# B&R Automation Studio project Embraco_PracoviskoPopisovaniaLaserom
Automation Studio 4.7.6.114 SP; technology packages: mapp 5.13.1

## Configuration Config1

CPU X20CP0484, AutomationRuntime D4.73, Build 6.3.0, Safety 1.10, Vc V4.72.4

### Task classes (Cpu.sw)
```
Cyclic#1 (cycle 2000 us, tolerance 0 us):
  CheckerKom <- Komunikacia_Checker.CheckerKomunikacia.prg
  MeranieTak <- Program.MeranieTaktime.prg
Cyclic#3 (cycle 50000 us, tolerance 50000 us):
  VstupnyOdd <- Program.VstupnyOddelovac.prg
  Popisovani <- Program.Popisovanie.prg
  Checker <- Program.Checker.prg
Cyclic#4 (cycle 100000 us, tolerance 100000 us):
  Main <- Program.Main.prg
  Poruchy_Si <- Program.Poruchy_Signalizacie.prg
  OvladanieG <- HMI.OvladanieGrafiky.prg
  Vycitanie_ <- Komunikacia_Laser.Vycitanie_casu.prg
  Ethernetov <- Komunikacia_Laser.EthernetovaKomunikacia.prg
Cyclic#5 (cycle 200000 us, tolerance 200000 us):
  Receptury <- Receptury.Receptury.prg
  Prihlasova <- PrihlasovaciSystem.PrihlasovaciSystem.prg
  Blikanie20 <- Blikace.Blikanie200ms.prg
Cyclic#6 (cycle 500000 us, tolerance 500000 us):
  Blikanie50 <- Blikace.Blikanie500ms.prg
Cyclic#7 (cycle 1000000 us, tolerance 1000000 us):
  Blikanie1s <- Blikace.Blikanie1s.prg
DataObjects: assl1
VcDataObjects: Visu <- HMI.Visu.dob
Binaries: vcfile, vcnet, vcbclass, vcfntttf, Visu01, arsvcreg, vcshared, vcpkat, vcpfgen, TCData, vcmgr, vctcal, vcalarm, vcdsloc, vcpdsw, vcdsint, vcrt, arial, udbdef, vcgclass, vcpdvnc, Visu02, vccdt, vccbmp, vccstr, vccbtn, vccline, vcclbox, arialbd, vccnum, vccalarm, vccbar, vcctext, Visu03, vccovl, vccshape, vcchspot, asnxdb1, iomap, Config_2, sysconf, Config, ashwac, Config_1, ashwd, asfw, User, arconfig, Role
Libraries: AsSafety, FileIO, DataObj, AsXml, standard, runtime, astime, AsBrStr, IecCheck, sys_lib, SC, MpRecipe, MpBase, AsTCP, AsMath, asieccon, vcresman
```

### Hardware
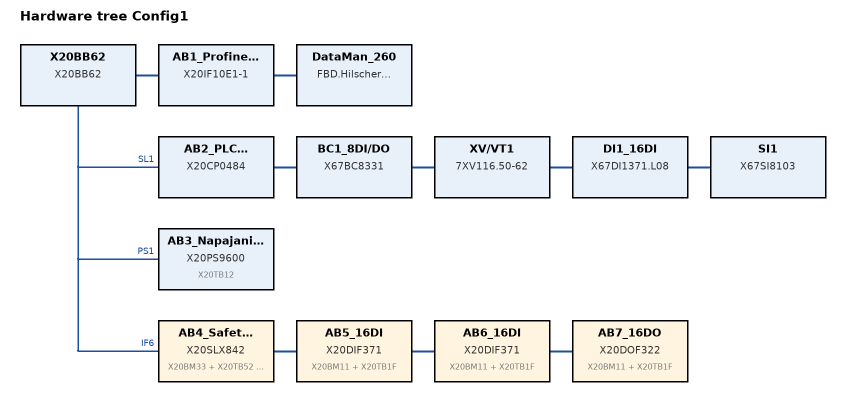
```
AB1_ProfinetMaster : X20IF10E1-1 v1.3.0.0  [SS -> X20BB62.SS1]
  Connector IF1:
    DtmRef = FBDIF.Hilscher.PNIOControllerDTM2.NETX 100 RE/PNM
    DtmId = eaec8113-ff32-47e2-8a6f-5691c0f842d4
  ConfigFile = AB1_ProfinetMaster.dtm
  ConfigModule = asnxdb1
AB2_PLC_X20CP0484 : X20CP0484 v1.4.2.0  [SL -> X20BB62.SL1]
  Connector IF2:
    ActivateDevice = 1
    Mode = Manual
    InternetAddress = 192.168.1.2
    SubnetMask = 255.255.255.0
    InaNodeNumber = 0
    Vnc1
    VncVcObjectName1 = Visu
    VncKeyMappingFile1 = VC\PS2-Keyboard.dis
    VncMaxConnections1 = 2
    VncRefreshRate1 = 100
  ConfigurationID = Embraco_PracoviskoPopisovaniaLaserom_Config1
  UserPartitionSize = 500
  UserRamSize = 10000
  RemMemSize = 20000
  PermanentPvSize = 8000
  TimerDeviceType = EPLX2X
  TimerDevice = AB2_PLC_X20CP0484.IF3
  TaskClassIdleTime = 2000
  Cyclic1Duration = 2000
  Cyclic1Tolerance = 0
  Cyclic2Duration = 10000
  Cyclic2Tolerance = 0
  Cyclic3Duration = 50000
  Cyclic3Tolerance = 50000
  Cyclic4Duration = 100000
  Cyclic4Tolerance = 100000
  Cyclic5Duration = 200000
  Cyclic5Tolerance = 200000
  Cyclic6Duration = 500000
  Cyclic6Tolerance = 500000
  Cyclic7Duration = 1000000
  Cyclic7Tolerance = 1000000
  Cyclic8Duration = 10000
  Cyclic8Tolerance = 30000000
  FileDevice1
  FileDeviceName1 = HDD
  FileDevicePath1 = F:\
  TimeZone = 145
  ActivateSntpServer = 1
  FtpUser1
  FtpUsername1 = admin
  FtpUserPassword1 = ZFxZtXmikHeuYrBmUWmLP4sX8b0VA9Bjt2tGuquGkoo=
  FtpUserSalt1 = qbFABSSZ
  FTPAccessRight1 = 0
AB3_NapajaniePLC : X20PS9600 v1.5.0.0  [PS -> X20BB62.PS1; SS1 -> X20TB12.SS]
AB4_SafetyMaster : X20SLX842 v1.10.12.1  [SS1 -> X20TB52.SS; SS2 -> X20TB52a.SS; SL -> X20BM33.SL1]
  Supervision = off
  SafeProject = SafeLOGIC-1
  SafeDesigner = 4.4.0.0
  DigitalOutput01 = viaSafeLOGIC
  DigitalOutput02 = viaSafeLOGIC
  DigitalOutput03 = viaSafeLOGIC
  DigitalOutput04 = viaSafeLOGIC
  DigitalOutput05 = viaSafeLOGIC
  DigitalOutput06 = viaSafeLOGIC
  UnsafeOutputBOOLs = 32
  UnsafeInputBOOLs = 32
AB5_16DI : X20DIF371 v1.1.0.0  [SS1 -> X20TB1F.SS; SL -> X20BM11.SL1]
  Supervision = off
AB6_16DI : X20DIF371 v1.1.0.0  [SS1 -> X20TB1F1.SS; SL -> X20BM11a.SL1]
  Supervision = off
AB7_16DO : X20DOF322 v1.4.0.0  [SS1 -> X20TB1F2.SS; SL -> X20BM11b.SL1]
  Supervision = off
BC1_8DI/DO : X67BC8331 v2.11.1.0  [PLK1 -> AB2_PLC_X20CP0484.IF3 [Cable Type=PowerlinkCable, Length=10, Version=1.0.0.2]]
DI1_16DI : X67DI1371.L08 v1.1.0.0  [X2X1 -> XV/VT1.X2X2 [Cable Type=X2XCable, Length=10, Version=1.0.0.2]]
  Supervision = off
DataMan_260 : FBD.Hilscher.PNIOGenDevDTM2.DataMan 260 v5.5.0 (OrderNumber=DataMan 260, VendorAddress=dataman)  [PN1 -> AB1_ProfinetMaster.IF1]
  DtmId = 4941676e-6e57-439f-abc9-d0f1f6497b10
  ChannelBlocks_47615121-fe6e-4591-b3b6-8465b3212ca9  // Acquisition Control <Slot 1>
  IO_OutputImage_47615121-fe6e-4591-b3b6-8465b3212ca9  // 1 Byte(s)
  ChannelBlocks_d194d4db-42e7-41e5-a767-b87b0401a075  // Acquisition Status <Slot 2>
  IO_InputImage_d194d4db-42e7-41e5-a767-b87b0401a075  // 3 Byte(s)
  ChannelBlocks_1f3ce926-3699-4ff7-ae20-f41f99e8e1a7  // Results Control <Slot 3>
  IO_OutputImage_1f3ce926-3699-4ff7-ae20-f41f99e8e1a7  // 1 Byte(s)
  ChannelBlocks_275960ff-423a-4b85-9ae8-7b4c1d1c8472  // Results Status <Slot 4>
  IO_InputImage_275960ff-423a-4b85-9ae8-7b4c1d1c8472  // 1 Byte(s)
  ChannelBlocks_ec76be99-af22-40a4-a52c-c51730de08a4  // Soft Event Control <Slot 5>
  IO_InputImage_ec76be99-af22-40a4-a52c-c51730de08a4  // 1 Byte(s)
  IO_OutputImage_ec76be99-af22-40a4-a52c-c51730de08a4  // 1 Byte(s)
  ChannelBlocks_de08c721-900e-43fb-8e68-4cff8c152ca9  // User Data - 64 bytes <Slot 6>
  IO_OutputImage_de08c721-900e-43fb-8e68-4cff8c152ca9  // 68 Byte(s)
  ChannelBlocks_b5868303-eee8-413e-96c2-c1ebf3a28649  // Result Data - 64 bytes <Slot 7>
  IO_InputImage_b5868303-eee8-413e-96c2-c1ebf3a28649  // 72 Byte(s)
SI1 : X67SI8103 v1.10.12.0  [X2X1 -> DI1_16DI.X2X2 [Cable Type=X2XCable, Length=10, Version=1.0.0.2]]
  Supervision = off
X20BB62 : X20BB62 v1.1.1.0
X20BM11 : X20BM11 v1.0.0.1  [X2X1 -> X20BM33.X2X2]
X20BM11a : X20BM11 v1.0.0.1  [X2X1 -> X20BM11.X2X2]
X20BM11b : X20BM11 v1.0.0.1  [X2X1 -> X20BM11a.X2X2]
X20BM33 : X20BM33 v1.0.0.6  [X2X1 -> X20BB62.IF6]
X20TB12 : X20TB12 v1.0.0.0
X20TB1F : X20TB1F v1.0.0.0
X20TB1F1 : X20TB1F v1.0.0.0
X20TB1F2 : X20TB1F v1.0.0.0
X20TB52 : X20TB52 v1.0.0.2
X20TB52a : X20TB52 v1.0.0.2
XV/VT1 : 7XV116.50-62 v1.2.0.0  [X2X1 -> BC1_8DI/DO.IF1 [Cable Type=X2XCable, Length=10, Version=1.0.0.2]]
  Supervision = off
```

### Cpu.per - AB2_PLC_X20CP0484/Cpu.per
```iecst
VAR_CONFIG
	Stav_StatorPopisany AT %MX0; (* *)
END_VAR
```

### IoMap.iom - AB2_PLC_X20CP0484/IoMap.iom
```iecst
VAR_CONFIG
	Cyclic#1.Safety.IN.CS_Panel_KanalA AT %IX."AB4_SafetyMaster".SafeDigitalInput01;
	Cyclic#1.Safety.IN.CS_Panel_KanalB AT %IX."AB4_SafetyMaster".SafeDigitalInput02;
	Cyclic#1.Safety.IN.CS_Checker_KanalA AT %IX."AB4_SafetyMaster".SafeDigitalInput03;
	Cyclic#1.Safety.IN.CS_Checker_KanalB AT %IX."AB4_SafetyMaster".SafeDigitalInput04;
	Cyclic#1.Safety.IN.VyblokovanieZamkov_KanalA AT %IX."AB4_SafetyMaster".SafeDigitalInput05;
	Cyclic#1.Safety.IN.VyblokovanieZamkov_KanalB AT %IX."AB4_SafetyMaster".SafeDigitalInput06;
	Cyclic#1.Safety.OUT.Zona_CS AT %IX."AB4_SafetyMaster".PhysicalStateChannel01;
	Cyclic#1.Safety.OUT.Zona_VnutroBunky AT %IX."AB4_SafetyMaster".PhysicalStateChannel02;
	Cyclic#1.Safety.OUT.Zona_Laser AT %IX."AB4_SafetyMaster".PhysicalStateChannel03;
	Cyclic#1.Safety.OUT.Zona_ExternyCS_KanalA AT %IX."AB4_SafetyMaster".PhysicalStateChannel05;
	Cyclic#1.Safety.OUT.Zona_ExternyCS_KanalB AT %IX."AB4_SafetyMaster".PhysicalStateChannel06;
	Cyclic#1.Safety.RESET_ZonyCS AT %QX."AB4_SafetyMaster".BOOL101;
	Cyclic#1.Safety.RESET_ZonyLaser AT %QX."AB4_SafetyMaster".BOOL102;
	Cyclic#1.Safety.RESET_ZonyVnutroBunky AT %QX."AB4_SafetyMaster".BOOL103;
	Cyclic#1.Safety.IN.ZonaCS_SpatnaVezba AT %QX."AB4_SafetyMaster".BOOL104;
	Cyclic#1.Safety.IN.ZonaLaser_SpatnaVezba AT %QX."AB4_SafetyMaster".BOOL105;
	Cyclic#1.Safety.IN.ZonaVnutroBunky_SpatnaVezba AT %QX."AB4_SafetyMaster".BOOL106;
	Cyclic#1.Zariadenie.IN.TlakVzduchu_OK AT %QX."AB4_SafetyMaster".BOOL107;
	Cyclic#1.Safety.STAV.SafetyPLC_Nabehlo AT %IX."AB4_SafetyMaster".BOOL001;
	Cyclic#1.Safety.STAV.CS_Panel_Odblokov AT %IX."AB4_SafetyMaster".BOOL002;
	Cyclic#1.Safety.STAV.CS_Checker_Odblokov AT %IX."AB4_SafetyMaster".BOOL003;
	Cyclic#1.Safety.STAV.DvereBunky_Zamknute AT %IX."AB4_SafetyMaster".BOOL004;
	Cyclic#1.Safety.STAV.SnimacKrytuLasera_Aktivny AT %IX."AB4_SafetyMaster".BOOL005;
	Cyclic#1.Safety.STAV.SnimacStatorPodLaserom_Aktivny AT %IX."AB4_SafetyMaster".BOOL006;
	Cyclic#1.Safety.STAV.VyblokovanieZamkov_Aktivne AT %IX."AB4_SafetyMaster".BOOL007;
	Cyclic#1.Safety.STAV.ZonaCS_Aktivna AT %IX."AB4_SafetyMaster".BOOL008;
	Cyclic#1.Safety.STAV.ZonaLaser_Aktivna AT %IX."AB4_SafetyMaster".BOOL009;
	Cyclic#1.Safety.STAV.ZonaVnutroBunky_Aktivna AT %IX."AB4_SafetyMaster".BOOL010;
	Cyclic#1.Safety.IN.DvereBunky_KanalA AT %IX."SI1".SafeDigitalInput01;
	Cyclic#1.Safety.IN.DvereBunky_KanalB AT %IX."SI1".SafeDigitalInput02;
	Cyclic#1.Safety.IN.StatorPodLaserom_KanalA AT %IX."SI1".SafeDigitalInput03;
	Cyclic#1.Safety.IN.StatorPodLaserom_KanalB AT %IX."SI1".SafeDigitalInput04;
	Cyclic#1.Safety.IN.KrytLasera_KanalA AT %IX."SI1".SafeDigitalInput05;
	Cyclic#1.Safety.IN.KrytLasera_KanalB AT %IX."SI1".SafeDigitalInput06;
	Cyclic#1.Safety.OUT.DvereBunky_Zamkni AT %QX."SI1".DigitalOutput01;
	Cyclic#1.Zariadenie.IN.PrepatovaOchrana_OK AT %IX."AB5_16DI".DigitalInput01;
	Cyclic#1.Safety.IN.ZdvihZdvizky_SpatnaVezba AT %QX."AB4_SafetyMaster".BOOL108;
	Cyclic#1.Zariadenie.IN.NapajanieOdsavania_OK AT %IX."AB5_16DI".DigitalInput02;
	Cyclic#1.Zariadenie.IN.NapajanieLasera_OK AT %IX."AB5_16DI".DigitalInput03;
	Cyclic#1.Zariadenie.IN.TlacitkoSTART AT %IX."AB5_16DI".DigitalInput04;
	Cyclic#1.Zariadenie.IN.TlacitkoSTOP AT %IX."AB5_16DI".DigitalInput05;
	Cyclic#1.Zariadenie.IN.TlacitkoRESET_CS AT %IX."AB5_16DI".DigitalInput06;
	Cyclic#1.Zariadenie.IN.TlakVzduchu_OK AT %IX."AB5_16DI".DigitalInput07;
	Cyclic#1.Checker.IN.TlacitkoBANNER AT %IX."AB5_16DI".DigitalInput08;
	Cyclic#1.Safety.IN.ZdvihZdvizky_SpatnaVezba AT %IX."AB5_16DI".DigitalInput09;
	Cyclic#1.Safety.IN.ZonaCS_SpatnaVezba AT %IX."AB5_16DI".DigitalInput10;
	Cyclic#1.Safety.IN.ZonaVnutroBunky_SpatnaVezba AT %IX."AB5_16DI".DigitalInput11;
	Cyclic#1.Safety.IN.ZonaLaser_SpatnaVezba AT %IX."AB5_16DI".DigitalInput12;
	Cyclic#1.Popisovanie.IN.Laser_StavREADY AT %IX."AB5_16DI".DigitalInput13;
	Cyclic#1.Popisovanie.IN.Laser_StavEND AT %IX."AB5_16DI".DigitalInput14;
	Cyclic#1.Popisovanie.IN.Laser_StavBUSY AT %IX."AB5_16DI".DigitalInput15;
	Cyclic#1.Popisovanie.IN.Laser_STARTUP AT %IX."AB5_16DI".DigitalInput16;
	Cyclic#1.Popisovanie.IN.Laser_ALARM AT %IX."AB6_16DI".DigitalInput01;
	Cyclic#1.Checker.IN.Checker_OUT0 AT %IX."AB6_16DI".DigitalInput02;
	Cyclic#1.Checker.IN.Checker_OUT1 AT %IX."AB6_16DI".DigitalInput03;
	Cyclic#1.Checker.IN.Checker_OUT2 AT %IX."AB6_16DI".DigitalInput04;
	Cyclic#1.Checker.IN.Checker_OUT3 AT %IX."AB6_16DI".DigitalInput05;
	Cyclic#1.Popisovanie.OUT.Odsavanie_Start AT %QX."AB7_16DO".DigitalOutput01;
	Cyclic#1.Zariadenie.OUT.LED_Dvojtlacitka_StartStop AT %QX."AB7_16DO".DigitalOutput02;
	Cyclic#1.Zariadenie.OUT.LED_Tlacitka_RESET_CS AT %QX."AB7_16DO".DigitalOutput03;
	Cyclic#1.Checker.OUT.BANNER_ZelenaLED AT %QX."AB7_16DO".DigitalOutput04;
	Cyclic#1.Checker.OUT.BANNER_CervenaLED AT %QX."AB7_16DO".DigitalOutput05;
	Cyclic#1.Popisovanie.OUT.Laser_StartZnacenia AT %QX."AB7_16DO".DigitalOutput06;
	Cyclic#1.Popisovanie.OUT.Laser_ResetPoruchy AT %QX."AB7_16DO".DigitalOutput07;
	Cyclic#1.Checker.OUT.Checker_IN0 AT %QX."AB7_16DO".DigitalOutput08;
	Cyclic#1.Checker.OUT.Checker_IN1 AT %QX."AB7_16DO".DigitalOutput09;
	Cyclic#1.Zariadenie.OUT.Majak_CerveneSvetlo AT %QX."AB7_16DO".DigitalOutput12;
	Cyclic#1.Zariadenie.OUT.Majak_ZlteSvetlo AT %QX."AB7_16DO".DigitalOutput13;
	Cyclic#1.Zariadenie.OUT.Majak_ZeleneSvetlo AT %QX."AB7_16DO".DigitalOutput14;
	Cyclic#1.Zariadenie.OUT.Majak_Hukacka AT %QX."AB7_16DO".DigitalOutput15;
	Cyclic#1.Checker.IN.Stoper1_ZASUNUTY AT %IX."BC1_8DI/DO".IF1.ST1.DigitalInput01;
	Cyclic#1.Checker.IN.Stoper1_VYSUNUTY AT %IX."BC1_8DI/DO".IF1.ST1.DigitalInput02;
	Cyclic#1.Checker.IN.ZasobaPredStoprom1 AT %IX."BC1_8DI/DO".IF1.ST1.DigitalInput03;
	Cyclic#1.Checker.IN.Stoper2_ZASUNUTY AT %IX."BC1_8DI/DO".IF1.ST1.DigitalInput04;
	Cyclic#1.Checker.IN.Stoper2_VYSUNUTY AT %IX."BC1_8DI/DO".IF1.ST1.DigitalInput05;
	Cyclic#1.Checker.IN.Stoper2_PritomnostPaletky AT %IX."BC1_8DI/DO".IF1.ST1.DigitalInput06;
	Cyclic#1.Checker.IN.ZaplnenieVystupnejTrate AT %IX."BC1_8DI/DO".IF1.ST1.DigitalInput07 INVERSE;
	Cyclic#1.Checker.IN.Stoper2_PritomnostStatora AT %IX."BC1_8DI/DO".IF1.ST1.DigitalInput08;
	Cyclic#1.VstupnyOddelovac.IN.Stoper1_ZASUNUTY AT %IX."DI1_16DI".DigitalInput01;
	Cyclic#1.VstupnyOddelovac.IN.Stoper1_VYSUNUTY AT %IX."DI1_16DI".DigitalInput02;
	Cyclic#1.Checker.IN.Stoper1_PritomnostPaletky AT %IX."DI1_16DI".DigitalInput03;
	Cyclic#1.VstupnyOddelovac.IN.Stoper2_ZASUNUTY AT %IX."DI1_16DI".DigitalInput04;
	Cyclic#1.VstupnyOddelovac.IN.Stoper2_VYSUNUTY AT %IX."DI1_16DI".DigitalInput05;
	Cyclic#1.VstupnyOddelovac.IN.Stoper2_PritomnostPaletky AT %IX."DI1_16DI".DigitalInput06 INVERSE;
	Cyclic#1.Popisovanie.IN.StoperZdvizky_ZASUNUTY AT %IX."DI1_16DI".DigitalInput07;
	Cyclic#1.Popisovanie.IN.StoperZdvizky_VYSUNUTY AT %IX."DI1_16DI".DigitalInput08;
	Cyclic#1.Popisovanie.IN.StoperZdvizky_PritomnostPaletky AT %IX."DI1_16DI".DigitalInput09 INVERSE;
	Cyclic#1.Popisovanie.IN.StoperZdvizky_PritomnostStatora AT %IX."DI1_16DI".DigitalInput10 INVERSE;
	Cyclic#1.VstupnyOddelovac.OUT.Stoper1_VYSUN AT %QX."XV/VT1".DigitalOutput01;
	Cyclic#1.Zariadenie.STAV.KOM_Modul_BC1_OK AT %IX."BC1_8DI/DO".ModuleOk;
	Cyclic#1.Zariadenie.STAV.KOM_Checker_OK AT %IX."DataMan_260".ModuleOk;
	Cyclic#1.Zariadenie.STAV.KOM_Modul_DI1_OK AT %IX."DI1_16DI".ModuleOk;
	Cyclic#1.Zariadenie.STAV.KOM_Modul_XV_OK AT %IX."XV/VT1".ModuleOk;
	Cyclic#1.Zariadenie.STAV.KOM_Modul_SI1_OK AT %IX."SI1".ModuleOk;
	Cyclic#1.Safety.IN.DvereBunky_AktuatorVzamku AT %IX."SI1".DigitalInput01;
	Cyclic#1.VstupnyOddelovac.OUT.Stoper2_VYSUN AT %QX."XV/VT1".DigitalOutput02;
	Cyclic#1.Popisovanie.OUT.StoperZdvizky_VYSUN AT %QX."XV/VT1".DigitalOutput03;
	Cyclic#1.Checker.OUT.Stoper1_VYSUN AT %QX."XV/VT1".DigitalOutput04;
	Cyclic#1.Checker.OUT.Stoper2_VYSUN AT %QX."XV/VT1".DigitalOutput05;
	Cyclic#1.Checker.OUT.Stoper2_ZASUN AT %QX."XV/VT1".DigitalOutput12;
	Cyclic#1.Checker.OUT.Stoper1_ZASUN AT %QX."XV/VT1".DigitalOutput13;
	Cyclic#1.VstupnyOddelovac.OUT.Stoper1_ZASUN AT %QX."XV/VT1".DigitalOutput14;
	Cyclic#1.VstupnyOddelovac.OUT.Stoper2_ZASUN AT %QX."XV/VT1".DigitalOutput15;
	Cyclic#1.Popisovanie.OUT.StoperZdvizky_ZASUN AT %QX."XV/VT1".DigitalOutput16;
	Cyclic#1.Popisovanie.OUT.Zdvizku_ZASUN AT %QX."AB7_16DO".DigitalOutput10;
	Cyclic#1.Popisovanie.OUT.Zdvizku_VYSUN AT %QX."AB7_16DO".DigitalOutput11;
	Cyclic#1.Popisovanie.IN.Zdvizka_VYSUNUTA AT %IX."DI1_16DI".DigitalInput11;
	Cyclic#1.Popisovanie.IN.Zdvizka_ZASUNUTA AT %IX."DI1_16DI".DigitalInput12;
	Cyclic#1.Checker.COM.ControlWord AT %QB."DataMan_260".Module001_Acquisition_Control_Register;
	Cyclic#1.Checker.COM.StatusWord AT %IB."DataMan_260".Module002_Acquisition_Status_Register;
	Cyclic#1.Checker.COM.ResultStatus AT %IB."DataMan_260".Module004_Results_Status_Register;
	Cyclic#1.Checker.COM.ResultData AT %IW."DataMan_260".Module007_Result_Code;
	Cyclic#1.Checker.COM.ResultControl AT %QB."DataMan_260".Module003_Results_Control_Register;
END_VAR
```

- Safety project (password-protected, skipped)

### Config.mprecipexml - AB2_PLC_X20CP0484/mappServices/Config.mprecipexml
```
Element gUzivatelXmlLink (Type=mprecipexml)
```

### Config_1.mprecipexml - AB2_PLC_X20CP0484/mappServices/Config_1.mprecipexml
```
Element gRecipeXmlLink (Type=mprecipexml)
```

### Config_2.mprecipexml - AB2_PLC_X20CP0484/mappServices/Config_2.mprecipexml
```
Element gPremenneXmlLink (Type=mprecipexml)
```

## Logical view

Binary libraries used (declarations not repeated): operator, runtime, astime, AsIecCon, AsSafety, FileIO, DataObj, AsXml, standard, AsBrStr, sys_lib, AsTCP, AsMath, MpRecipe 5.13.1, MpBase 5.13.0

### Global.typ - Global data types
```iecst
(*************Vyčítavanie systémového času**********************)

TYPE
	Cas : 	STRUCT
		Hodina : USINT;
		Minuta : USINT;
		Sekunda : USINT;
	END_STRUCT;
	Datum : 	STRUCT
		Den : USINT;
		Mesiac : USINT;
		Rok : UINT;
	END_STRUCT;
	Cas_STR : 	STRUCT
		Hodina : STRING[2];
		Minuta : STRING[2];
		Sekunda : STRING[2];
	END_STRUCT;
	Datum_STR : 	STRUCT
		Den : STRING[2];
		Mesiac : STRING[2];
		Rok : STRING[2];
	END_STRUCT;
END_TYPE

(**************Ovládanie lasera**********************)

TYPE
	Client_typ : 	STRUCT  (*TCP Client Variables*)
		sStep : UINT; (*TCP Client Step Variable*)
		TcpOpen_0 : TcpOpen; (*AsTCP.TcpOpen FUB*)
		TcpClient_0 : TcpClient; (*AsTCP.TcpClient FUB*)
		TcpRecv_0 : TcpRecv; (*AsTCP.TcpRecv FUB*)
		TcpSend_0 : TcpSend; (*AsTCP.TcpSend FUB*)
		TcpIoctl_0 : TcpIoctl; (*AsTCP.TcpIoctl FUB*)
		TcpClose_0 : TcpClose; (*AsTCP.TcpClose FUB*)
		linger_opt : tcpLINGER_typ; (*AsTCP.tcpLINGER_typ*)
		recv_timeout : UDINT; (*receive timeout*)
		TcpOpen_timeout : UDINT;
		TcpClient_timeout : UDINT;
	END_STRUCT;
	Laser_typ : 	STRUCT
		Commands : LaserCommands_typ;
		Status : LaserStatus_typ;
		Data : LaserData_typ;
	END_STRUCT;
	LaserCommands_typ : 	STRUCT
		OdosliDataSpravy : BOOL;
		ResetPoruchy : BOOL;
		VyberSpravuLasera : BOOL;
	END_STRUCT;
	LaserStatus_typ : 	STRUCT
		PoruchaOtvoreniaKomunikacie : BOOL;
		PoruchaOdoslaniaDat : BOOL;
		PoruchaZatvoreniaKomunikacie : BOOL;
		PoruchaSpojenia_s_Laserom : BOOL;
		PoruchaPrijatiaDat : BOOL;
		OdoslanieDatSpravy_OK : BOOL;
		OdoslanieDatSpravy_NG : BOOL;
		VyberSpravy_OK : BOOL;
		VyberSpravy_NG : BOOL;
		StrataKomunikacie : BOOL;
		VysledokPorovnaniaOdpovede : DINT;
	END_STRUCT;
	LaserData_typ : 	STRUCT  (*Datatyp for global Variables*)
		Data : USINT;
	END_STRUCT;
END_TYPE

(***************Uzivatelia****************************)

TYPE
	ParametreUzivatelovTyp : 	STRUCT
		Meno : STRING[50];
		Heslo : STRING[50];
		UrovenUzivatela : UINT;
	END_STRUCT;
END_TYPE

(************Receptury*************************)

TYPE
	ParametreRecepturTyp : 	STRUCT
		NazovStatora : STRING[50];
		BOM_kod_Statora : STRING[20];
	END_STRUCT;
END_TYPE

(************Remanentne premenné*************)

TYPE
	RemPremenne_typ : 	STRUCT
		RemPrem_0 : UDINT;
	END_STRUCT;
END_TYPE

(**************Zariadenie************************)

TYPE
	Zariadenie_typ : 	STRUCT
		Automat : BOOL;
		Manual : BOOL;
		Reset : BOOL;
		KoniecCyklu : BOOL;
		KoniecModelu : BOOL;
		Hukacka_ON : BOOL;
		Hukacka_OFF : BOOL;
		IN : ZariadenieIN_typ;
		OUT : ZariadenieOUT_typ;
		PAR : ZariadeniePAR_typ;
		STAV : ZariadenieSTAV_typ;
		TaktTime_START : BOOL;
		TaktTime_RESET : BOOL;
		TaktTime_ZAPIS : BOOL;
		TaktTime_Milisekundy : UINT;
		TaktTime_Sekundy : UINT;
		TaktTime_Minuty : UINT;
		TaktTime_Hodiny : UINT;
		TaktTime_NameraneSekundy : UINT;
		TaktTime_NameraneMinuty : UINT;
		TaktTime_NameraneHodiny : UINT;
		PriechodnyRezim : BOOL;
	END_STRUCT;
	ZariadenieIN_typ : 	STRUCT
		PrepatovaOchrana_OK : BOOL;
		TlakVzduchu_OK : BOOL;
		NapajanieLasera_OK : BOOL;
		NapajanieOdsavania_OK : BOOL;
		TlacitkoSTART : BOOL;
		TlacitkoSTOP : BOOL;
		TlacitkoRESET_CS : BOOL;
	END_STRUCT;
	ZariadenieOUT_typ : 	STRUCT
		Majak_ZeleneSvetlo : BOOL;
		Majak_ZlteSvetlo : BOOL;
		Majak_CerveneSvetlo : BOOL;
		Majak_Hukacka : BOOL;
		LED_Dvojtlacitka_StartStop : BOOL;
		LED_Tlacitka_RESET_CS : BOOL;
	END_STRUCT;
	ZariadeniePAR_typ : 	STRUCT
		PAR_0 : UDINT;
	END_STRUCT;
	ZariadenieSTAV_typ : 	STRUCT
		Automat : BOOL;
		Manual : BOOL;
		PoINIT : BOOL;
		UkoncenieCyklu : BOOL;
		StavZariadenia : USINT;
		KOM_Checker_OK : BOOL;
		KOM_Modul_BC1_OK : BOOL;
		KOM_Modul_SI1_OK : BOOL;
		KOM_Modul_DI1_OK : BOOL;
		KOM_Modul_XV_OK : BOOL;
		Moduly_OK : BOOL;
		TlakVzduchuOK : BOOL;
		PrebiehaResetPoruchy : BOOL;
		NezvolenaReceptura : BOOL;
	END_STRUCT;
END_TYPE

(*************Vstupný oddelovač***************)

TYPE
	VstupnyOddelovac_typ : 	STRUCT
		Automat : BOOL;
		Manual : BOOL;
		Reset : BOOL;
		KoniecCyklu : BOOL;
		IN : VstupnyOddelovacIN_typ;
		OUT : VstupnyOddelovacOUT_typ;
		PAR : VstupnyOddelovacPAR_typ;
		STAV : VstupnyOddelovacSTAV_typ;
	END_STRUCT;
	VstupnyOddelovacIN_typ : 	STRUCT
		Stoper1_ZASUNUTY : BOOL;
		Stoper1_VYSUNUTY : BOOL;
		Stoper2_ZASUNUTY : BOOL;
		Stoper2_VYSUNUTY : BOOL;
		Stoper2_PritomnostPaletky : BOOL;
	END_STRUCT;
	VstupnyOddelovacOUT_typ : 	STRUCT
		Stoper1_VYSUN : BOOL;
		Stoper1_ZASUN : BOOL;
		Stoper2_VYSUN : BOOL;
		Stoper2_ZASUN : BOOL;
	END_STRUCT;
	VstupnyOddelovacPAR_typ : 	STRUCT
		PAR_0 : UDINT;
	END_STRUCT;
	VstupnyOddelovacSTAV_typ : 	STRUCT
		PoINIT : BOOL;
		Stopre_PoziciaNAVAZANIE : BOOL;
		Stopre_PoziciaVYVAZANIE : BOOL;
	END_STRUCT;
END_TYPE

(*************Popisovanie***************)

TYPE
	Popisovanie_typ : 	STRUCT
		Automat : BOOL;
		Manual : BOOL;
		Reset : BOOL;
		KoniecCyklu : BOOL;
		IN : PopisovanieIN_typ;
		OUT : PopisovanieOUT_typ;
		PAR : PopisovaniePAR_typ;
		STAV : PopisovanieSTAV_typ;
	END_STRUCT;
	PopisovanieIN_typ : 	STRUCT
		Laser_StavREADY : BOOL;
		Laser_StavEND : BOOL;
		Laser_StavBUSY : BOOL;
		Laser_STARTUP : BOOL;
		Laser_ALARM : BOOL;
		StoperZdvizky_ZASUNUTY : BOOL;
		StoperZdvizky_VYSUNUTY : BOOL;
		StoperZdvizky_PritomnostPaletky : BOOL;
		StoperZdvizky_PritomnostStatora : BOOL;
		Zdvizka_VYSUNUTA : BOOL;
		Zdvizka_ZASUNUTA : BOOL;
	END_STRUCT;
	PopisovanieOUT_typ : 	STRUCT
		Odsavanie_Start : BOOL;
		Laser_StartZnacenia : BOOL;
		Laser_ResetPoruchy : BOOL;
		Zdvizku_VYSUN : BOOL;
		Zdvizku_ZASUN : BOOL;
		StoperZdvizky_ZASUN : BOOL;
		StoperZdvizky_VYSUN : BOOL;
	END_STRUCT;
	PopisovaniePAR_typ : 	STRUCT
		PocetPrazdnychPaletiek : USINT;
	END_STRUCT;
	PopisovanieSTAV_typ : 	STRUCT
		PoINIT : BOOL;
		Zdvizka_PritomnostNGkusu : BOOL;
	END_STRUCT;
END_TYPE

(*************Checker***************)

TYPE
	Checker_typ : 	STRUCT
		Automat : BOOL;
		Manual : BOOL;
		Reset : BOOL;
		KoniecCyklu : BOOL;
		IN : CheckerIN_typ;
		OUT : CheckerOUT_typ;
		COM : CheckerCOM_typ;
		PAR : CheckerPAR_typ;
		STAV : CheckerSTAV_typ;
		TRIGER_Enable : BOOL;
		TRIGER : BOOL;
		Vysledok_POTVRDENIE : BOOL;
		KAMERA_OFF : BOOL;
	END_STRUCT;
	CheckerIN_typ : 	STRUCT
		TlacitkoBANNER : BOOL;
		Checker_OUT0 : BOOL; (*OUT_0*)
		Checker_OUT1 : BOOL; (*OUT_1*)
		Checker_OUT2 : BOOL; (*OUT_2*)
		Checker_OUT3 : BOOL; (*OUT_3*)
		Stoper1_ZASUNUTY : BOOL;
		Stoper1_VYSUNUTY : BOOL;
		Stoper2_ZASUNUTY : BOOL;
		Stoper2_VYSUNUTY : BOOL;
		ZasobaPredStoprom1 : BOOL;
		Stoper1_PritomnostPaletky : BOOL;
		Stoper2_PritomnostPaletky : BOOL;
		Stoper2_PritomnostStatora : BOOL;
		ZaplnenieVystupnejTrate : BOOL;
	END_STRUCT;
	CheckerOUT_typ : 	STRUCT
		BANNER_ZelenaLED : BOOL;
		BANNER_CervenaLED : BOOL;
		Checker_IN0 : BOOL;
		Checker_IN1 : BOOL;
		Stoper1_VYSUN : BOOL;
		Stoper1_ZASUN : BOOL;
		Stoper2_VYSUN : BOOL;
		Stoper2_ZASUN : BOOL;
	END_STRUCT;
	CheckerCOM_typ : 	STRUCT
		ControlWord : USINT;
		StatusWord : USINT;
		ResultStatus : USINT;
		ResultControl : USINT;
		ResultData : UINT;
	END_STRUCT;
	CheckerPAR_typ : 	STRUCT
		PAR_0 : UDINT;
	END_STRUCT;
	CheckerSTAV_typ : 	STRUCT
		PoINIT : BOOL;
		Stopre_PoziciaNAVAZANIE : BOOL;
		Stopre_PoziciaVYVAZANIE : BOOL;
		TRIGER_Ready : BOOL;
		BUSY : BOOL;
		Vysledok_READY : BOOL;
		Vysledok_OK : BOOL;
		Vysledok_NG : BOOL;
	END_STRUCT;
END_TYPE

(**************Bezpecnost************************)

TYPE
	Safety_typ : 	STRUCT
		IN : SafetyIN_typ;
		OUT : SafetyOUT_typ;
		PAR : SafetyPAR_typ;
		STAV : SafetySTAV_typ;
		RESET_ZonyLaser : BOOL;
		RESET_ZonyVnutroBunky : BOOL;
		RESET_ZonyCS : BOOL;
		OdomkniDvereBunky : BOOL;
	END_STRUCT;
	SafetyIN_typ : 	STRUCT
		DvereBunky_AktuatorVzamku : BOOL;
		ZonaCS_SpatnaVezba : BOOL;
		ZonaLaser_SpatnaVezba : BOOL;
		ZonaVnutroBunky_SpatnaVezba : BOOL;
		DvereBunky_KanalA : BOOL;
		DvereBunky_KanalB : BOOL;
		CS_Panel_KanalA : BOOL;
		CS_Panel_KanalB : BOOL;
		CS_Checker_KanalA : BOOL;
		CS_Checker_KanalB : BOOL;
		VyblokovanieZamkov_KanalA : BOOL;
		VyblokovanieZamkov_KanalB : BOOL;
		ExternyCS_KanalA : BOOL;
		ExternyCS_KanalB : BOOL;
		StatorPodLaserom_KanalA : BOOL;
		StatorPodLaserom_KanalB : BOOL;
		KrytLasera_KanalA : BOOL;
		KrytLasera_KanalB : BOOL;
		ZdvihZdvizky_SpatnaVezba : BOOL;
	END_STRUCT;
	SafetyOUT_typ : 	STRUCT
		Zona_CS : BOOL; (*SO1*)
		Zona_VnutroBunky : BOOL; (*SO3*)
		Zona_Laser : BOOL;
		Zona_ExternyCS_KanalA : BOOL;
		Zona_ExternyCS_KanalB : BOOL;
		DvereBunky_Zamkni : BOOL;
	END_STRUCT;
	SafetyPAR_typ : 	STRUCT
		PAR_0 : USINT;
	END_STRUCT;
	SafetySTAV_typ : 	STRUCT
		SafetyPLC_Nabehlo : BOOL;
		CS_Checker_Odblokov : BOOL;
		CS_Panel_Odblokov : BOOL;
		ZonaCS_Aktivna : BOOL;
		ZonaLaser_Aktivna : BOOL;
		ZonaVnutroBunky_Aktivna : BOOL;
		VyblokovanieZamkov_Aktivne : BOOL;
		SnimacKrytuLasera_Aktivny : BOOL;
		SnimacStatorPodLaserom_Aktivny : BOOL;
		DvereBunky_Zamknute : BOOL;
	END_STRUCT;
END_TYPE

(**************Vizualizacia************************)

TYPE
	Vizualizacia_typ : 	STRUCT
		Slider : USINT;
		CisloAktualnejObrazovky : USINT;
		CisloZadanejObrazovky : USINT;
		LED_TlacitkaResetCS : USINT;
		LED_TlacitkaZamokDveriBunky : USINT;
		BlikanieTlacitkaSTART : BOOL;
		ZamkniTlacitkoRezimAutomat : USINT;
		ZamkniTlacitkoRezimManual : USINT;
		ZamkniTlacitkoSTART : USINT;
		ZamkniTlacitkoSTOP : USINT;
		ZamkniTlacitkoZamokDveriBunky : USINT;
		ZamkniTlacitkaOvladaniaZdvizky : USINT;
		ZamkniTlacitkoPriechodnyRezim : USINT;
		ZamkniTlacitkoLaserVolbaSpravy : USINT;
		ZamkniTlacitkoLaserPosliData : USINT;
		Zobraz_ResetZariadenia : USINT;
		Zobraz_HlasenieOdoberStator : USINT;
		Zobraz_HlasenieZamkyVyblokovane : USINT;
		Zobraz_HlasenieNezvolenaRecept : USINT;
		Zobraz_HlasenieNizkyTlakVzduchu : USINT;
		Zobraz_HlasenieVymenaModelu : USINT;
		Zobraz_HlasenieNaZdvizkeNGkus : USINT;
		Zobraz_TlacitkoOK_ZmenaModelu : USINT;
		Stav_VystupnyOddelovac : USINT;
		Stav_Laser : USINT;
		Stav_Checker : USINT;
		TlacitkoZamkniDvereBunky : BOOL;
		TlacitkoRezimAutomat : BOOL;
		ZamkniTlacitko_StartPopisovania : USINT;
		ZamkniTlacitko_PriechodnyRezim : USINT;
	END_STRUCT;
	QRkod_typ : 	STRUCT
		BOM_Statora : STRING[7];
		DatumVyroby : STRING[6];
		CasVyroby : STRING[6];
		NazovVyrobnejLinky : STRING[8];
		BOM_PosledneZnaky : STRING[4];
	END_STRUCT;
END_TYPE
```

### Global.var - Global variables
```iecst
(************Vyčítavanie systémového času************************)
VAR
	Zapnutie_citania_casu : BOOL;
	System_Cas_Datum : DTStructure;
	Status_citania_casu : UINT;
	Systemovy_Cas : Cas;
	Systemovy_Datum : Datum;
	Systemovy_Cas_STR : Cas_STR;
	Systemovy_Datum_STR : Datum_STR;
END_VAR
VAR CONSTANT
	SeparatorCasu : STRING[1] := ':';
	SeparatorDatumu : STRING[1] := '.';
END_VAR
VAR
	TextPole_Cas : STRING[6];
	TextPole_Datum : STRING[6];
	Sekunda_String : STRING[2];
	Hodina_String : STRING[2];
	Minuta_String : STRING[2];
	Mesiac_String : STRING[2];
	Den_String : STRING[2];
END_VAR
(************Ovládanie Komunikácie s laserom*******************)
VAR
	Client : Client_typ;
	Laser : Laser_typ;
	Laser_DataSpravy : ARRAY[0..47] OF USINT := [2,4,65,1,41,11(0),1,7(0),2,7(0),3,9(0),4,4(0),3];
	Laser_NazovSpravy : ARRAY[0..12] OF USINT := [2,10,87,0,108,105,110,2(101),109,2(0),3];
	Laser_Sprava : ARRAY[0..50] OF USINT;
	Laser_Odpoved : ARRAY[0..50] OF USINT;
	OK_OdpovedNaDataSpravy : ARRAY[0..50] OF USINT := [240,2(32),55,57,127,2(48),56,48,2,4,65,1,6,0,5,5(1),3,28(0)];
	OK_OdpovedNaVyberSpravy : ARRAY[0..50] OF USINT := [240,2(32),55,57,127,2(48),56,48,2(2),87,0,3,36(0)];
END_VAR
(**********Blikače*******************************)
VAR
	Blikac200ms : BOOL;
	Blikac500ms : BOOL;
	Blikac5s : BOOL;
	Blikac1s : BOOL;
END_VAR
(*****************Alarmy*************************)
VAR
	Alarmy : ARRAY[0..100] OF BOOL;
	NastalaPorucha : BOOL;
	ZobrazSymbolAlarmu : BOOL;
	PotvrdenieAlarmov : BOOL;
	PoruchaVstupnehoOddelovaca : BOOL;
	PoruchaPopisovania : BOOL;
	PoruchaCheckera : BOOL;
END_VAR
(*************Premenne receptur**************)
VAR
	MpRecipeRegPar_0 : MpRecipeRegPar := (0);
	MpRecipeXml_0 : MpRecipeXml := (0);
	Receptura : ARRAY[0..150] OF ParametreRecepturTyp := [151((0))];
	ZoznamReceptur : ARRAY[0..150] OF STRING[50] := [151('')];
	UlozRecepturu : BOOL := FALSE;
	NacitajRecepturu : BOOL;
	NazovStatora : STRING[50] := '';
	BOM_kod_Statora : STRING[7];
	ZvolenyNazovStatora : STRING[50];
	ZvolenyBOM_kod_Statora : STRING[7];
END_VAR
(**********Premenne uzivatelov********************************)
VAR
	MpRecipeXml_1 : MpRecipeXml := (0);
	MpRecipeRegPar_1 : MpRecipeRegPar := (0);
	Uzivatel : ARRAY[0..50] OF ParametreUzivatelovTyp;
	ZoznamUzivatelov : ARRAY[0..50] OF STRING[50] := [51('')];
	MenoUzivatela : STRING[50];
	HesloUzivatela : STRING[50];
	UrovenUzivatela : UINT;
	ZadaneMenoUzivatela : STRING[50];
	ZadaneHesloUzivatela : STRING[50];
	ZvolenyUzivatel : STRING[50];
	ZvolenaUroven : UINT;
	TP_ZobrazPopUpPrihlasenie : USINT;
	UlozUzivatelov : BOOL;
	PrihlasUzivatela : BOOL;
	VymazUzivatela : BOOL;
	OdhlasUzivatela : BOOL;
	SC_Uzivatelia : SequenceControlTyp;
END_VAR
(************Všeobecné premenné********************************)
VAR
	Safety : Safety_typ;
	Vizu : Vizualizacia_typ;
	Zariadenie : Zariadenie_typ;
	SC_VstupnyOddelovac : SequenceControlTyp;
	VstupnyOddelovac : VstupnyOddelovac_typ;
	SC_Popisovanie : SequenceControlTyp;
	Popisovanie : Popisovanie_typ;
	SC_Checker : SequenceControlTyp;
	Checker : Checker_typ;
	QR_Kod : QRkod_typ;
END_VAR
VAR RETAIN
	Stav_StatorPopisany : BOOL;
END_VAR
```

### Package Logical/Libraries - Global libraries

### Library Logical/Libraries/IecCheck (IEC)
Depends on: sys_lib, AsBrStr

#### IecCheck.fun - Exported functions and function blocks
```iecst
FUNCTION CheckDivSint : SINT (* Check divisor for SINT division *)
	VAR_INPUT
		divisor : SINT;
	END_VAR
END_FUNCTION

FUNCTION CheckDivUsint : USINT (* Check divisor for USINT division *)
	VAR_INPUT
		divisor : USINT;
	END_VAR
END_FUNCTION

FUNCTION CheckDivInt : INT (* Check divisor for INT division *)
	VAR_INPUT
		divisor : INT;
	END_VAR
END_FUNCTION

FUNCTION CheckDivUint : UINT (* Check divisor for UINT division *)
	VAR_INPUT
		divisor : UINT;
	END_VAR
END_FUNCTION

FUNCTION CheckDivDint : DINT (* Check divisor for DINT division *)
	VAR_INPUT
		divisor : DINT;
	END_VAR
END_FUNCTION

FUNCTION CheckDivUdint : UDINT (* Check divisor for UDINT division *)
	VAR_INPUT
		divisor : UDINT;
	END_VAR
END_FUNCTION

FUNCTION CheckDivReal : REAL (* Check divisor for REAL division *)
	VAR_INPUT
		divisor : REAL;
	END_VAR
END_FUNCTION

FUNCTION CheckDivLReal : LREAL (* Check divisor for LREAL division, not available for SG3 and SGC *)
	VAR_INPUT
		divisor : LREAL;
	END_VAR
END_FUNCTION

FUNCTION CheckBounds : DINT (* Check range for array access *)
	VAR_INPUT
		index : DINT;
		lower : DINT;
		upper : DINT;
	END_VAR
END_FUNCTION

FUNCTION CheckRange : DINT (* Check range for enumeration *)
	VAR_INPUT
		value : DINT;
		lower : DINT;
		upper : DINT;
	END_VAR
END_FUNCTION

FUNCTION CheckSignedSubrange : DINT (* Check range for subrange of signed data types *)
	VAR_INPUT
		value : DINT;
		lower : DINT;
		upper : DINT;
	END_VAR
END_FUNCTION

FUNCTION CheckUnsignedSubrange : UDINT (* Check range for subrange of unsigned data types *)
	VAR_INPUT
		value : UDINT;
		lower : UDINT;
		upper : UDINT;
	END_VAR
END_FUNCTION

FUNCTION CheckReadAccess : UDINT (* Check address when reading dynamic variables *)
	VAR_INPUT
		address : UDINT;
	END_VAR
END_FUNCTION

FUNCTION CheckWriteAccess : UDINT (* Check address when writing dynamic variables *)
	VAR_INPUT
		address : UDINT;
	END_VAR
END_FUNCTION

FUNCTION MakeEntry : UDINT (* Makes an entry (log book entry) in the error log book *)
	VAR
		taskname : STRING[30];
		group : USINT;
		status_name : UINT;
		out_text : STRING[80];
	END_VAR
	VAR_INPUT
		number : UINT;
		index : DINT;
		text : STRING[50];
	END_VAR
END_FUNCTION
```

#### IecCheck.st - Implementation file
```iecst
(* Check divisor for SINT division *)
FUNCTION CheckDivSint
	IF divisor=0 THEN
		CheckDivSint:=1;
		MakeEntry(55555,divisor,'CheckDivSint');
	ELSE
		CheckDivSint:=divisor;
	END_IF
END_FUNCTION

(* Check divisor for USINT division *)
FUNCTION CheckDivUsint
	IF divisor=0 THEN
		CheckDivUsint:=1;
		MakeEntry(55555,divisor,'CheckDivUsint');
	ELSE
		CheckDivUsint:=divisor;
	END_IF
END_FUNCTION

(* Check divisor for INT division *)
FUNCTION CheckDivInt
	IF divisor=0 THEN
		CheckDivInt:=1;
		MakeEntry(55555,divisor,'CheckDivInt');
	ELSE
		CheckDivInt:=divisor;
	END_IF
END_FUNCTION

(* Check divisor for UINT division *)
FUNCTION CheckDivUint
	IF divisor=0 THEN
		CheckDivUint:=1;
		MakeEntry(55555,divisor,'CheckDivUint');
	ELSE
		CheckDivUint:=divisor;
	END_IF
END_FUNCTION

(* Check divisor for DINT division *)
FUNCTION CheckDivDint
	IF divisor=0 THEN
		CheckDivDint:=1;
		MakeEntry(55555,divisor,'CheckDivDint');
	ELSE
		CheckDivDint:=divisor;
	END_IF
END_FUNCTION

(* Check divisor for UDINT division *)
FUNCTION CheckDivUdint
	IF divisor=0 THEN
		CheckDivUdint:=1;
		MakeEntry(55555,divisor,'CheckDivUdint');
	ELSE
		CheckDivUdint:=divisor;
	END_IF
END_FUNCTION

(* Check divisor for REAL division *)
FUNCTION CheckDivReal
	IF divisor=0 THEN
		CheckDivReal:=1;
		MakeEntry(55555,0,'CheckDivReal');
	ELSE
		CheckDivReal:=divisor;
	END_IF
END_FUNCTION

(* Check divisor for LREAL division *)
FUNCTION CheckDivLReal
	IF divisor=0 THEN
		CheckDivLReal:=1;
		MakeEntry(55555,0,'CheckDivLReal');
	ELSE
		CheckDivLReal:=divisor;
	END_IF
END_FUNCTION

(* Check range for array access *)
FUNCTION CheckBounds
	IF index < lower THEN
		CheckBounds := lower;
		MakeEntry(55555,index,'CheckBounds');
	ELSIF index > upper THEN
		CheckBounds := upper;
		MakeEntry(55555,index,'CheckBounds');
	ELSE
		CheckBounds := index;
	END_IF
END_FUNCTION

(* Check range for enumeration *)
FUNCTION CheckRange
	IF value < lower THEN
		CheckRange := lower;
		MakeEntry(55555,value,'CheckRange');
	ELSIF value > upper THEN
		CheckRange := upper;
		MakeEntry(55555,value,'CheckRange');
	ELSE
		CheckRange := value;
	END_IF
END_FUNCTION

(* Check range for subrange of signed data types *)
FUNCTION CheckSignedSubrange
	IF value < lower THEN
		CheckSignedSubrange := lower;
		MakeEntry(55555,value,'CheckSignedSubrange');
	ELSIF value > upper THEN
		CheckSignedSubrange := upper;
		MakeEntry(55555,value,'CheckSignedSubrange');
	ELSE
		CheckSignedSubrange := value;
	END_IF
END_FUNCTION

(* Check range for subrange of unsigned data types *)
FUNCTION CheckUnsignedSubrange
	IF value < lower THEN
		CheckUnsignedSubrange := lower;
		MakeEntry(55555,value,'CheckUnsignedSubrange');
	ELSIF value > upper THEN
		CheckUnsignedSubrange := upper;
		MakeEntry(55555,value,'CheckUnsignedSubrange');
	ELSE
		CheckUnsignedSubrange := value;
	END_IF
END_FUNCTION

(* Check address when reading dynamic variables *)
FUNCTION CheckReadAccess
	IF address=0 THEN
		(* TODO: Insert an appropriate code, see AutomationStudio help for further information *)
		MakeEntry(55555,address,'Read from NULL');
	END_IF

	CheckReadAccess:=0;
END_FUNCTION

(* Check address when writing dynamic variables *)
FUNCTION CheckWriteAccess
	IF address=0 THEN
		(* TODO: Insert an appropriate code, see AutomationStudio help for further information *)
		MakeEntry(55555,address,'Write to NULL');
	END_IF

	CheckWriteAccess:=0;
END_FUNCTION

(* Makes an entry (log book entry) in the error log book *)
FUNCTION MakeEntry
		status_name := ST_name(0,ADR(taskname),ADR(group));

		brsstrcpy(ADR(out_text),ADR(text));
		brsstrcat(ADR(out_text),ADR(' > in task > '));
  		brsstrcat(ADR(out_text),ADR(taskname));
		MakeEntry := ADR(out_text);
		ERRxfatal(number,index,ADR(out_text));
END_FUNCTION
```

### Library Logical/Libraries/SC (IEC)

#### Types.typ - Exported data types
```iecst
TYPE
	SequenceControlTyp : 	STRUCT
		StepName : STRING[80];
		Step : UINT;
		Switch1 : BOOL;
		Switch2 : BOOL;
		Switch3 : BOOL;
		ResetStep : BOOL;
		LastStep : BOOL;
		IdleTime : TON;
		AlarmTime : TON;
	END_STRUCT;
END_TYPE
```

#### SC.fun - Exported functions and function blocks
```iecst
FUNCTION SequenceControl : BOOL
	VAR_IN_OUT
		SC : SequenceControlTyp;
	END_VAR
END_FUNCTION
```

#### SequenceControl.st
```iecst
(* TODO: Add your comment here *)
FUNCTION SequenceControl

	IF SC.ResetStep THEN
		brsmemset(ADR(SC.StepName),0,SIZEOF(SC.StepName));
		SC.Switch1:= FALSE;
		SC.Switch2:= FALSE;
		SC.Switch3:= FALSE;
		SC.IdleTime.IN:= FALSE;
		SC.AlarmTime.IN:= FALSE;
		SC.ResetStep:= FALSE;
	END_IF

	IF SC.LastStep THEN
		brsmemset(ADR(SC.StepName),0,SIZEOF(SC.StepName));
		SC.Switch1:= FALSE;
		SC.Switch2:= FALSE;
		SC.Switch3:= FALSE;
		SC.IdleTime.IN:= FALSE;
		SC.AlarmTime.IN:= FALSE;
		SC.Step:= 0;
		SC.LastStep:= FALSE;
	END_IF

	//Volanie časovačov//
	SC.AlarmTime();
	SC.IdleTime();

END_FUNCTION
```

### Program Logical/Program/Main (IEC)

#### Main.st - Init, cyclic, exit code
```iecst
PROGRAM _INIT
	(* Insert code here *)

END_PROGRAM

PROGRAM _CYCLIC

	//Volanie podprogramov//
	OvlSafety;

	//Zariadenie stav Automat//
	IF VstupnyOddelovac.Automat OR Popisovanie.Automat OR Checker.Automat THEN
		Zariadenie.STAV.Automat:= TRUE;
	ELSE
		Zariadenie.STAV.Automat:= FALSE;
		Zariadenie.STAV.UkoncenieCyklu:= FALSE;
	END_IF

	//Zariadenie stav Manual//
	IF VstupnyOddelovac.Manual OR Popisovanie.Manual OR Checker.Manual THEN
		Zariadenie.STAV.Manual:= TRUE;
	ELSE
		Zariadenie.STAV.Manual:= FALSE;
	END_IF

	//Zariadenie stav po inicializacii//
	IF VstupnyOddelovac.STAV.PoINIT AND Popisovanie.STAV.PoINIT AND Checker.STAV.PoINIT THEN
		Zariadenie.STAV.PoINIT:= TRUE;
	ELSE
		Zariadenie.STAV.PoINIT:= FALSE;
	END_IF

	//Spustenie režimu automat//
	IF EDGEPOS(Zariadenie.IN.TlacitkoSTART)THEN
		IF Safety.STAV.ZonaCS_Aktivna AND NOT NastalaPorucha AND Safety.STAV.ZonaVnutroBunky_Aktivna AND NOT Zariadenie.STAV.UkoncenieCyklu AND Zariadenie.IN.TlakVzduchu_OK AND NOT Zariadenie.STAV.Manual AND Zariadenie.STAV.Moduly_OK AND Vizu.CisloAktualnejObrazovky = 2 AND NOT Zariadenie.STAV.NezvolenaReceptura AND NOT Zariadenie.KoniecModelu THEN
			VstupnyOddelovac.Automat:= TRUE;
			Popisovanie.Automat:= TRUE;
			Checker.Automat:= TRUE;
		END_IF
	END_IF

	//Spustenie režimu manual//
	IF Zariadenie.Manual THEN
		IF Safety.STAV.ZonaCS_Aktivna AND NOT NastalaPorucha AND NOT Zariadenie.STAV.Automat THEN
			VstupnyOddelovac.Manual:= TRUE;
			Popisovanie.Manual:= TRUE;
			Checker.Manual:= TRUE;
		END_IF
		Zariadenie.Manual:= FALSE;
	END_IF

	//Resetovanie zariadenia pri stlačení tlačítka režim automat//
	IF Vizu.TlacitkoRezimAutomat THEN
		IF NOT Zariadenie.STAV.Automat THEN
			Zariadenie.Reset:= TRUE;
		END_IF
		Vizu.TlacitkoRezimAutomat:= FALSE;
	END_IF

	//Reset zariadenia//
	IF Zariadenie.Reset THEN
		VstupnyOddelovac.Reset:= TRUE;
		Popisovanie.Reset:= TRUE;
		Checker.Reset:= TRUE;
		Zariadenie.Reset:= FALSE;
	END_IF

	//Resetovanie zariadenia pri stlačení tlačítka režim automat//
	IF Vizu.TlacitkoRezimAutomat THEN
		IF NOT Zariadenie.STAV.Automat THEN
			Zariadenie.Reset:= TRUE;
		END_IF
		Vizu.TlacitkoRezimAutomat:= FALSE;
	END_IF

	//Ukončenie cyklu zariadenia//
	IF EDGEPOS(Zariadenie.IN.TlacitkoSTOP) OR Zariadenie.KoniecCyklu THEN
		IF Zariadenie.STAV.PoINIT AND NOT Zariadenie.STAV.UkoncenieCyklu THEN
			VstupnyOddelovac.KoniecCyklu:= TRUE;
			Popisovanie.KoniecCyklu:= TRUE;
			Checker.KoniecCyklu:= TRUE;
			Zariadenie.STAV.UkoncenieCyklu:= TRUE;
		END_IF
		Zariadenie.KoniecCyklu:= FALSE;
	END_IF

	//Stav externé moduly OK//
	Zariadenie.STAV.Moduly_OK:= Zariadenie.STAV.KOM_Modul_BC1_OK AND Zariadenie.STAV.KOM_Modul_DI1_OK AND Zariadenie.STAV.KOM_Modul_SI1_OK AND Zariadenie.STAV.KOM_Modul_XV_OK (*AND Zariadenie.STAV.KOM_Checker_OK*);

	//Príznak nezvolená receptura//
	IF ZvolenyNazovStatora = '' AND NOT Zariadenie.PriechodnyRezim THEN
		Zariadenie.STAV.NezvolenaReceptura:= TRUE;
		Vizu.Zobraz_HlasenieNezvolenaRecept:= 0;
	ELSE
		Zariadenie.STAV.NezvolenaReceptura:= FALSE;
		Vizu.Zobraz_HlasenieNezvolenaRecept:= 1;
	END_IF

END_PROGRAM

PROGRAM _EXIT
	(* Insert code here *)

END_PROGRAM
```

#### OvlSafety.st
```iecst
ACTION OvlSafety:

	//********************************************Ovladanie zámkov****************************************************//
	//Zámok dverí bunky//
	IF EDGEPOS(Vizu.TlacitkoZamkniDvereBunky) THEN
		IF Safety.STAV.ZonaCS_Aktivna AND Safety.IN.DvereBunky_AktuatorVzamku AND NOT Safety.STAV.DvereBunky_Zamknute AND Zariadenie.IN.TlakVzduchu_OK THEN
			Safety.OUT.DvereBunky_Zamkni:= TRUE;
		ELSIF Safety.STAV.DvereBunky_Zamknute AND NOT Zariadenie.STAV.Automat THEN
			Safety.OUT.DvereBunky_Zamkni:= FALSE;
		END_IF
	ELSIF NOT Safety.STAV.ZonaCS_Aktivna THEN
		Safety.OUT.DvereBunky_Zamkni:= FALSE;
	ELSIF Safety.OdomkniDvereBunky AND NOT Zariadenie.STAV.Automat THEN
		Safety.OUT.DvereBunky_Zamkni:= FALSE;
	END_IF

	IF NOT Safety.STAV.DvereBunky_Zamknute THEN
		Safety.OdomkniDvereBunky:= FALSE;
	END_IF

	//****************************************Resetovanie zón****************************************************************//
	//Reset zóny CS//
	Safety.RESET_ZonyCS:= Zariadenie.IN.TlacitkoRESET_CS;

	//Reset zóny vnútra bunky//
	IF Safety.STAV.ZonaCS_Aktivna AND Safety.STAV.DvereBunky_Zamknute AND NOT Safety.STAV.ZonaVnutroBunky_Aktivna THEN
		Safety.RESET_ZonyVnutroBunky:= TRUE;
	ELSE
		Safety.RESET_ZonyVnutroBunky:= FALSE;
	END_IF

	//Reset zóny laser//
	IF Safety.STAV.ZonaCS_Aktivna AND Safety.STAV.ZonaVnutroBunky_Aktivna AND Safety.STAV.SnimacKrytuLasera_Aktivny AND Safety.STAV.SnimacStatorPodLaserom_Aktivny AND NOT Safety.STAV.ZonaLaser_Aktivna THEN
		Safety.RESET_ZonyLaser:= TRUE;
	ELSE
		Safety.RESET_ZonyLaser:= FALSE;
	END_IF

END_ACTION
```

### Program Logical/Program/VstupnyOddelovac (IEC)

#### Main.st - Init, cyclic, exit code
```iecst
PROGRAM _INIT
	(* Insert code here *)

END_PROGRAM

PROGRAM _CYCLIC

	//Volanie podprogramov//
	OvlStoprov;

	//Volanie funkcie SequenceControl//
	SequenceControl(SC:= SC_VstupnyOddelovac);

	//Reset sekcie //
	IF VstupnyOddelovac.Reset OR PoruchaVstupnehoOddelovaca THEN
		SC_VstupnyOddelovac.Step:= 0;
	END_IF

	CASE SC_VstupnyOddelovac.Step OF

		0:
			SC_VstupnyOddelovac.StepName:='0 - Nulovanie';
			SC_OvlStoprov.Step:= 0;
			VstupnyOddelovac.Automat:= FALSE;
			VstupnyOddelovac.KoniecCyklu:= FALSE;
			VstupnyOddelovac.Manual:= FALSE;
			VstupnyOddelovac.Reset:= FALSE;
			VstupnyOddelovac.STAV.PoINIT:= FALSE;

			IF Safety.STAV.ZonaCS_Aktivna AND NOT PoruchaVstupnehoOddelovaca AND Zariadenie.IN.TlakVzduchu_OK THEN
				SC_VstupnyOddelovac.ResetStep:= TRUE;
				SC_VstupnyOddelovac.Step:= 1;
			END_IF

		1:
			SC_VstupnyOddelovac.StepName:='1 - Cakam na spustenie vyroby';
			IF VstupnyOddelovac.Automat THEN
				SC_VstupnyOddelovac.Step:= 2;
			ELSIF VstupnyOddelovac.Manual THEN
				SC_VstupnyOddelovac.Step:= 700;
			END_IF

		//********************************************************Inicializácia****************************************************************************//

		2:
			SC_VstupnyOddelovac.StepName:='2 - Inicializacia - cakam na spustenie inicializacie';
			SC_VstupnyOddelovac.IdleTime.PT:= T#500ms;
			SC_VstupnyOddelovac.AlarmTime.PT:= T#5s;

			SC_VstupnyOddelovac.IdleTime.IN:= TRUE;

			IF SC_VstupnyOddelovac.IdleTime.Q THEN
				SC_VstupnyOddelovac.ResetStep:= TRUE;
				SC_VstupnyOddelovac.Step:= 3;
			END_IF

		3:
			SC_VstupnyOddelovac.StepName:='3 - Inicializacia - rozhodnutie o inicializacii';
			SC_VstupnyOddelovac.IdleTime.PT:= T#500ms;
			SC_VstupnyOddelovac.AlarmTime.PT:= T#5s;

			IF VstupnyOddelovac.STAV.Stopre_PoziciaNAVAZANIE THEN
				VstupnyOddelovac.STAV.PoINIT:= TRUE;
				SC_VstupnyOddelovac.ResetStep:= TRUE;
				SC_VstupnyOddelovac.Step:= 100;
			ELSIF VstupnyOddelovac.STAV.Stopre_PoziciaVYVAZANIE THEN
				SC_VstupnyOddelovac.ResetStep:= TRUE;
				SC_VstupnyOddelovac.Step:= 5;
			ELSE
				SC_VstupnyOddelovac.ResetStep:= TRUE;
				SC_VstupnyOddelovac.Step:= 5;
			END_IF

		5:
			SC_VstupnyOddelovac.StepName:='5 - Inicializacia - cakam na odchod paletky z 2 stopra';
			SC_VstupnyOddelovac.IdleTime.PT:= T#1s;
			SC_VstupnyOddelovac.AlarmTime.PT:= T#5s;

			SC_VstupnyOddelovac.IdleTime.IN:= NOT VstupnyOddelovac.IN.Stoper2_PritomnostPaletky;

			IF SC_VstupnyOddelovac.IdleTime.Q THEN
				SC_VstupnyOddelovac.ResetStep:= TRUE;
				SC_VstupnyOddelovac.Step:= 7;
			END_IF

		7:
			SC_VstupnyOddelovac.StepName:='7 - Inicializacia - preklopenie stoprov do pozicie navazania';
			SC_VstupnyOddelovac.IdleTime.PT:= T#500ms;
			SC_VstupnyOddelovac.AlarmTime.PT:= T#5s;

			IF NOT SC_VstupnyOddelovac.Switch1 THEN
				Stopre_pozNAVAZANIE:= TRUE;
				SC_VstupnyOddelovac.Switch1:= TRUE;
			END_IF

			IF VstupnyOddelovac.STAV.Stopre_PoziciaNAVAZANIE THEN
				VstupnyOddelovac.STAV.PoINIT:= TRUE;
				SC_VstupnyOddelovac.ResetStep:= TRUE;
				SC_VstupnyOddelovac.Step:= 100;
			END_IF

		//********************************************************Automatický režim****************************************************************************//

		100:
			SC_VstupnyOddelovac.StepName:='100 - Automaticky Rezim - cakam na pritomnost paletky na 2 stopri a vyvezenie na stoper zdvizky';
			SC_VstupnyOddelovac.IdleTime.PT:= T#100ms;
			SC_VstupnyOddelovac.AlarmTime.PT:= T#5s;

			SC_VstupnyOddelovac.IdleTime.IN:= NOT Popisovanie.IN.StoperZdvizky_PritomnostPaletky;

			IF VstupnyOddelovac.KoniecCyklu THEN
				SC_VstupnyOddelovac.ResetStep:= TRUE;
				SC_VstupnyOddelovac.Step:= 0;
			ELSIF Zariadenie.KoniecModelu THEN
				SC_VstupnyOddelovac.ResetStep:= TRUE;
				SC_VstupnyOddelovac.Step:= 0;
			ELSIF Popisovanie.STAV.PoINIT THEN
				IF VstupnyOddelovac.IN.Stoper2_PritomnostPaletky AND Popisovanie.IN.Zdvizka_ZASUNUTA AND Popisovanie.IN.StoperZdvizky_VYSUNUTY AND NOT Popisovanie.IN.StoperZdvizky_PritomnostPaletky THEN
					SC_VstupnyOddelovac.ResetStep:= TRUE;
					SC_VstupnyOddelovac.Step:= 101;
				ELSIF VstupnyOddelovac.IN.Stoper2_PritomnostPaletky AND Popisovanie.IN.Zdvizka_ZASUNUTA AND SC_VstupnyOddelovac.IdleTime.Q THEN
					SC_VstupnyOddelovac.ResetStep:= TRUE;
					SC_VstupnyOddelovac.Step:= 101;
				END_IF
			END_IF

		101:
			SC_VstupnyOddelovac.StepName:='101 - Automaticky Rezim - preklopenie stoprov do pozicie vyvazania';
			SC_VstupnyOddelovac.IdleTime.PT:= T#500ms;
			SC_VstupnyOddelovac.AlarmTime.PT:= T#5s;

			IF NOT SC_VstupnyOddelovac.Switch1 THEN
				Stopre_pozVYVAZANIE:= TRUE;
				SC_VstupnyOddelovac.Switch1:= TRUE;
			END_IF

			IF VstupnyOddelovac.STAV.Stopre_PoziciaVYVAZANIE THEN
				SC_VstupnyOddelovac.ResetStep:= TRUE;
				SC_VstupnyOddelovac.Step:= 105;
			END_IF

		105:
			SC_VstupnyOddelovac.StepName:='105 - Automaticky Rezim - cakam na odchod paletky z 2 stopra';
			SC_VstupnyOddelovac.IdleTime.PT:= T#500ms;
			SC_VstupnyOddelovac.AlarmTime.PT:= T#5s;

			SC_VstupnyOddelovac.IdleTime.IN:= NOT VstupnyOddelovac.IN.Stoper2_PritomnostPaletky;

			IF SC_VstupnyOddelovac.IdleTime.Q THEN
				SC_VstupnyOddelovac.ResetStep:= TRUE;
				SC_VstupnyOddelovac.Step:= 108;
			END_IF

		108:
			SC_VstupnyOddelovac.StepName:='108 - Automaticky Rezim - preklopenie stoprov do pozicie navazania';
			SC_VstupnyOddelovac.IdleTime.PT:= T#500ms;
			SC_VstupnyOddelovac.AlarmTime.PT:= T#5s;

			IF NOT SC_VstupnyOddelovac.Switch1 THEN
				Stopre_pozNAVAZANIE:= TRUE;
				SC_VstupnyOddelovac.Switch1:= TRUE;
			END_IF

			IF VstupnyOddelovac.STAV.Stopre_PoziciaNAVAZANIE THEN
				SC_VstupnyOddelovac.ResetStep:= TRUE;
				SC_VstupnyOddelovac.Step:= 100;
			END_IF

			//*******************************************************Manuálny režim*******************************************************************************//
		700:
			SC_VstupnyOddelovac.StepName:='700 - Manualny Rezim';
			SC_VstupnyOddelovac.IdleTime.PT:= T#8s;
			SC_VstupnyOddelovac.AlarmTime.PT:= T#5s;

	END_CASE

END_PROGRAM

PROGRAM _EXIT
	(* Insert code here *)

END_PROGRAM
```

#### Variables.var - Local variables
```iecst
VAR
	SC_OvlStoprov : SequenceControlTyp;
	Stopre_pozNAVAZANIE : BOOL;
	Stopre_pozVYVAZANIE : BOOL;
END_VAR
```

#### OvlStoprov.st
```iecst
ACTION OvlStoprov:

	//Pozice stoprov//
	VstupnyOddelovac.STAV.Stopre_PoziciaNAVAZANIE:= VstupnyOddelovac.IN.Stoper1_ZASUNUTY AND VstupnyOddelovac.IN.Stoper2_VYSUNUTY;
	VstupnyOddelovac.STAV.Stopre_PoziciaVYVAZANIE:= VstupnyOddelovac.IN.Stoper1_VYSUNUTY AND VstupnyOddelovac.IN.Stoper2_ZASUNUTY;

	//Volanie funkcie SequenceControl//
	SequenceControl(SC:= SC_OvlStoprov);

	CASE SC_OvlStoprov.Step OF

		0:
			SC_OvlStoprov.StepName:= '0 - Nulovanie';
			Stopre_pozNAVAZANIE:= FALSE;
			Stopre_pozVYVAZANIE:= FALSE;
			VstupnyOddelovac.OUT.Stoper1_VYSUN:= FALSE;
			VstupnyOddelovac.OUT.Stoper1_ZASUN:= FALSE;
			VstupnyOddelovac.OUT.Stoper2_VYSUN:= FALSE;
			VstupnyOddelovac.OUT.Stoper2_ZASUN:= FALSE;
			IF SC_VstupnyOddelovac.Step <> 0 THEN
				SC_OvlStoprov.ResetStep:= TRUE;
				SC_OvlStoprov.Step:= 1;
			END_IF

		1:
			SC_OvlStoprov.StepName:= '1 - Rozhodnutie o cinnosti';
			IF Stopre_pozNAVAZANIE THEN
				SC_OvlStoprov.Step:= 10;
			ELSIF Stopre_pozVYVAZANIE THEN
				SC_OvlStoprov.Step:= 20;
			END_IF

		10:
			SC_OvlStoprov.StepName:= '10 - Prepnutie oddelovaca do pozicie navazania';
			SC_OvlStoprov.IdleTime.PT:= T#3s;
			SC_OvlStoprov.AlarmTime.PT:= T#3s;

			IF VstupnyOddelovac.Automat THEN
				SC_OvlStoprov.AlarmTime.IN:= TRUE;
			ELSE
				SC_OvlStoprov.IdleTime.IN:= TRUE;
			END_IF

			IF NOT SC_OvlStoprov.Switch1 THEN
				VstupnyOddelovac.OUT.Stoper1_ZASUN:= TRUE;
				VstupnyOddelovac.OUT.Stoper2_VYSUN:= TRUE;
				SC_OvlStoprov.Switch1:= TRUE;
			END_IF

			IF SC_OvlStoprov.AlarmTime.Q THEN
				IF NOT VstupnyOddelovac.IN.Stoper1_ZASUNUTY THEN
					Alarmy[11]:= TRUE;
				ELSIF NOT VstupnyOddelovac.IN.Stoper2_VYSUNUTY THEN
					Alarmy[14]:= TRUE;
				END_IF
				PoruchaVstupnehoOddelovaca:= TRUE;
				Zariadenie.KoniecCyklu:= TRUE;
			END_IF

			IF VstupnyOddelovac.STAV.Stopre_PoziciaNAVAZANIE OR SC_OvlStoprov.IdleTime.Q THEN
				SC_OvlStoprov.ResetStep:= TRUE;
				SC_OvlStoprov.Step:= 0;
			END_IF

		20:
			SC_OvlStoprov.StepName:= '20 - Prepnutie oddelovaca do pozicie vyvazania';
			SC_OvlStoprov.IdleTime.PT:= T#3s;
			SC_OvlStoprov.AlarmTime.PT:= T#3s;

			IF VstupnyOddelovac.Automat THEN
				SC_OvlStoprov.AlarmTime.IN:= TRUE;
			ELSE
				SC_OvlStoprov.IdleTime.IN:= TRUE;
			END_IF

			IF NOT SC_OvlStoprov.Switch1 THEN
				VstupnyOddelovac.OUT.Stoper1_VYSUN:= TRUE;
				VstupnyOddelovac.OUT.Stoper2_ZASUN:= TRUE;
				SC_OvlStoprov.Switch1:= TRUE;
			END_IF

			IF SC_OvlStoprov.AlarmTime.Q THEN
				IF NOT VstupnyOddelovac.IN.Stoper1_VYSUNUTY THEN
					Alarmy[13]:= TRUE;
				ELSIF NOT VstupnyOddelovac.IN.Stoper2_ZASUNUTY THEN
					Alarmy[12]:= TRUE;
				END_IF
				PoruchaVstupnehoOddelovaca:= TRUE;
				Zariadenie.KoniecCyklu:= TRUE;
			END_IF

			IF VstupnyOddelovac.STAV.Stopre_PoziciaVYVAZANIE OR SC_OvlStoprov.IdleTime.Q THEN
				SC_OvlStoprov.ResetStep:= TRUE;
				SC_OvlStoprov.Step:= 0;
			END_IF

	END_CASE

END_ACTION
```

### Program Logical/Program/Popisovanie (IEC)

#### Main.st - Init, cyclic, exit code
```iecst
PROGRAM _INIT
	(* Insert code here *)

END_PROGRAM

PROGRAM _CYCLIC

	//Volanie podprogramov//
	OvlStopra;
	OvlZdvizky;
	SpravaPreLaser;

	//Volanie funkcie SequenceControl//
	SequenceControl(SC:= SC_Popisovanie);

	//Reset sekcie //
	IF Popisovanie.Reset OR PoruchaPopisovania THEN
		SC_Popisovanie.Step:= 0;
	END_IF

	CASE SC_Popisovanie.Step OF

		0:
			SC_Popisovanie.StepName:='0 - Nulovanie';
			SC_OvlStopra.Step:= 0;
			SC_OvlZdvizky.Step:= 0;
			Popisovanie.Automat:= FALSE;
			Popisovanie.KoniecCyklu:= FALSE;
			Popisovanie.Manual:= FALSE;
			Popisovanie.Reset:= FALSE;
			Popisovanie.STAV.PoINIT:= FALSE;
			Laser.Commands.VyberSpravuLasera:= FALSE;
			Laser.Commands.OdosliDataSpravy:= FALSE;
			Popisovanie.OUT.Laser_StartZnacenia:= FALSE;
			Popisovanie.OUT.Odsavanie_Start:= FALSE;
			Popisovanie.PAR.PocetPrazdnychPaletiek:= 0;
			Popisovanie.STAV.Zdvizka_PritomnostNGkusu:= FALSE;

			IF Safety.STAV.ZonaCS_Aktivna AND NOT PoruchaPopisovania AND Zariadenie.IN.TlakVzduchu_OK AND Safety.STAV.ZonaVnutroBunky_Aktivna THEN
				SC_Popisovanie.ResetStep:= TRUE;
				SC_Popisovanie.Step:= 1;
			END_IF

		1:
			SC_Popisovanie.StepName:='1 - Cakam na spustenie vyroby';
			IF Popisovanie.Automat THEN
				SC_Popisovanie.Step:= 2;
			ELSIF Popisovanie.Manual THEN
				SC_Popisovanie.Step:= 700;
			END_IF

			//********************************************************Inicializácia****************************************************************************//

		2:
			SC_Popisovanie.StepName:='2 - Inicializacia - cakam na spustenie inicializacie';
			SC_Popisovanie.IdleTime.PT:= T#500ms;
			SC_Popisovanie.AlarmTime.PT:= T#5s;

			SC_Popisovanie.IdleTime.IN:= TRUE;

			IF SC_Popisovanie.IdleTime.Q THEN
				Zariadenie.TaktTime_RESET:= TRUE;
				SC_Popisovanie.ResetStep:= TRUE;
				SC_Popisovanie.Step:= 3;
			END_IF

		3:
			SC_Popisovanie.StepName:='3 - Inicializacia - rozhodnutie o inicializacii';
			SC_Popisovanie.IdleTime.PT:= T#500ms;
			SC_Popisovanie.AlarmTime.PT:= T#5s;

			IF Popisovanie.IN.Zdvizka_ZASUNUTA THEN
				IF Popisovanie.IN.StoperZdvizky_VYSUNUTY THEN
					SC_Popisovanie.ResetStep:= TRUE;
					SC_Popisovanie.Step:= 15;
				ELSIF Popisovanie.IN.StoperZdvizky_ZASUNUTY THEN
					SC_Popisovanie.ResetStep:= TRUE;
					SC_Popisovanie.Step:= 4;
				END_IF
			ELSE
				IF Popisovanie.IN.StoperZdvizky_VYSUNUTY THEN
					SC_Popisovanie.ResetStep:= TRUE;
					SC_Popisovanie.Step:= 10;
				ELSIF Popisovanie.IN.StoperZdvizky_ZASUNUTY THEN
					SC_Popisovanie.ResetStep:= TRUE;
					SC_Popisovanie.Step:= 5;
				END_IF
			END_IF

		4:
			SC_Popisovanie.StepName:='4 - Inicializacia - cakam na odchod paletky zo stopra zdvizky';
			SC_Popisovanie.IdleTime.PT:= T#1s;
			SC_Popisovanie.AlarmTime.PT:= T#5s;

			SC_Popisovanie.IdleTime.IN:= NOT Popisovanie.IN.StoperZdvizky_PritomnostPaletky;

			IF SC_Popisovanie.IdleTime.Q THEN
				SC_Popisovanie.ResetStep:= TRUE;
				SC_Popisovanie.Step:= 5;
			END_IF

		5:
			SC_Popisovanie.StepName:='5 - Inicializacia - vysunutie stopra zdvizky';
			SC_Popisovanie.IdleTime.PT:= T#500ms;
			SC_Popisovanie.AlarmTime.PT:= T#5s;

			IF NOT SC_Popisovanie.Switch1 THEN
				StoperZdvizky_VYSUN:= TRUE;
				SC_Popisovanie.Switch1:= TRUE;
			END_IF

			IF Popisovanie.IN.StoperZdvizky_VYSUNUTY THEN
				SC_Popisovanie.ResetStep:= TRUE;
				SC_Popisovanie.Step:= 10;
			END_IF

		10:
			SC_Popisovanie.StepName:='10 - Inicializacia - zasunutie zdvizky';
			SC_Popisovanie.IdleTime.PT:= T#500ms;
			SC_Popisovanie.AlarmTime.PT:= T#5s;

			IF NOT SC_Popisovanie.Switch1 THEN
				Zdvizku_ZASUN:= TRUE;
				SC_Popisovanie.Switch1:= TRUE;
			END_IF

			IF Popisovanie.IN.Zdvizka_ZASUNUTA THEN
				SC_Popisovanie.ResetStep:= TRUE;
				SC_Popisovanie.Step:= 15;
			END_IF

		15:
			SC_Popisovanie.StepName:='15 - Inicializacia - vyber spravy do lasera';
			SC_Popisovanie.IdleTime.PT:= T#500ms;
			SC_Popisovanie.AlarmTime.PT:= T#5s;

			IF NOT SC_Popisovanie.Switch1 THEN
				Laser.Commands.VyberSpravuLasera:= TRUE;
				SC_Popisovanie.Switch1:= TRUE;
			END_IF

			IF EDGEPOS(Laser.Status.VyberSpravy_OK) THEN
				Popisovanie.STAV.PoINIT:= TRUE;
				IF NOT Zariadenie.PriechodnyRezim THEN
					Popisovanie.OUT.Odsavanie_Start:= TRUE;
				END_IF
				SC_Popisovanie.ResetStep:= TRUE;
				SC_Popisovanie.Step:= 100;
			ELSIF EDGEPOS(Laser.Status.VyberSpravy_NG) THEN
				Alarmy[29]:= TRUE;
				PoruchaPopisovania:= TRUE;
				Zariadenie.KoniecCyklu:= TRUE;
			END_IF

			//********************************************************Automatický režim****************************************************************************//

		100:
			SC_Popisovanie.StepName:='100 - Automaticky Rezim - cakam na pritomnost paletky na stopri zdvizky';
			SC_Popisovanie.IdleTime.PT:= T#500ms;
			SC_Popisovanie.AlarmTime.PT:= T#5s;

			SC_Popisovanie.IdleTime.IN:= Popisovanie.IN.StoperZdvizky_PritomnostPaletky;

			IF Popisovanie.KoniecCyklu THEN
				SC_Popisovanie.ResetStep:= TRUE;
				SC_Popisovanie.Step:= 0;
			ELSIF Zariadenie.KoniecModelu THEN
				SC_Popisovanie.ResetStep:= TRUE;
				SC_Popisovanie.Step:= 0;
			ELSIF SC_Popisovanie.IdleTime.Q THEN
				SC_Popisovanie.ResetStep:= TRUE;
				SC_Popisovanie.Step:= 103;
			END_IF

		103:
			SC_Popisovanie.StepName:='103 - Automaticky Rezim - rozhodnutie o popisovani statora';
			SC_Popisovanie.IdleTime.PT:= T#8s;
			SC_Popisovanie.AlarmTime.PT:= T#5s;

			IF Zariadenie.PriechodnyRezim THEN
				SC_Popisovanie.ResetStep:= TRUE;
				SC_Popisovanie.Step:= 130;
			ELSIF Stav_StatorPopisany THEN
				SC_Popisovanie.ResetStep:= TRUE;
				SC_Popisovanie.Step:= 130;
			ELSIF Popisovanie.IN.StoperZdvizky_PritomnostStatora THEN
				Popisovanie.PAR.PocetPrazdnychPaletiek:= 0;
				SC_Popisovanie.ResetStep:= TRUE;
				SC_Popisovanie.Step:= 105;
			ELSE
				Popisovanie.PAR.PocetPrazdnychPaletiek:= Popisovanie.PAR.PocetPrazdnychPaletiek + 1;
				SC_Popisovanie.ResetStep:= TRUE;
				SC_Popisovanie.Step:= 120;
			END_IF

		105:
			SC_Popisovanie.StepName:='105 - Automaticky Rezim - kontrola safety snimaca statora pod laserom';
			SC_Popisovanie.IdleTime.PT:= T#8s;
			SC_Popisovanie.AlarmTime.PT:= T#5s;

			IF NOT Safety.STAV.SnimacStatorPodLaserom_Aktivny THEN
				Zariadenie.TaktTime_ZAPIS:= TRUE;
				Zariadenie.TaktTime_START:= TRUE;
				SC_Popisovanie.ResetStep:= TRUE;
				SC_Popisovanie.Step:= 107;
			ELSE
				Alarmy[23]:= TRUE;
				PoruchaPopisovania:= TRUE;
				Zariadenie.KoniecCyklu:= TRUE;
			END_IF

		107:
			SC_Popisovanie.StepName:='107 - Automaticky Rezim - vysunutie zdvizky';
			SC_Popisovanie.IdleTime.PT:= T#8s;
			SC_Popisovanie.AlarmTime.PT:= T#4s;

			IF NOT SC_Popisovanie.Switch1 THEN
				Zdvizku_VYSUN:= TRUE;
				SC_Popisovanie.AlarmTime.IN:= TRUE;
				SC_Popisovanie.Switch1:= TRUE;
			END_IF

			IF Safety.STAV.SnimacStatorPodLaserom_Aktivny THEN
				SC_Popisovanie.ResetStep:= TRUE;
				SC_Popisovanie.Step:= 111;
			ELSIF SC_Popisovanie.AlarmTime.Q THEN
				Popisovanie.STAV.Zdvizka_PritomnostNGkusu:= TRUE;
				SC_Popisovanie.ResetStep:= TRUE;
				SC_Popisovanie.Step:= 110;
			END_IF

		110:
			SC_Popisovanie.StepName:='107 - Automaticky Rezim - cakam na potvrdenie obsluhy';
			SC_Popisovanie.IdleTime.PT:= T#8s;
			SC_Popisovanie.AlarmTime.PT:= T#5s;

			IF NOT Popisovanie.STAV.Zdvizka_PritomnostNGkusu AND SC_OvlZdvizky.Step = 1 THEN
				SC_Popisovanie.ResetStep:= TRUE;
				SC_Popisovanie.Step:= 115;
			END_IF

		111:
			SC_Popisovanie.StepName:='111 - Automaticky Rezim - posielam spravu do lasera';
			SC_Popisovanie.IdleTime.PT:= T#8s;
			SC_Popisovanie.AlarmTime.PT:= T#5s;

			IF NOT SC_Popisovanie.Switch1 THEN
				Laser.Commands.OdosliDataSpravy:= TRUE;
				SC_Popisovanie.Switch1:= TRUE;
			END_IF

			IF EDGEPOS(Laser.Status.OdoslanieDatSpravy_OK) THEN
				SC_Popisovanie.ResetStep:= TRUE;
				SC_Popisovanie.Step:= 112;
			ELSIF EDGEPOS(Laser.Status.OdoslanieDatSpravy_NG) THEN
				Alarmy[26]:= TRUE;
				PoruchaPopisovania:= TRUE;
				Zariadenie.KoniecCyklu:= TRUE;
			END_IF

		112:
			SC_Popisovanie.StepName:='112 - Automaticky Rezim - cakam na stav Laser READY';
			SC_Popisovanie.IdleTime.PT:= T#8s;
			SC_Popisovanie.AlarmTime.PT:= T#5s;

			SC_Popisovanie.AlarmTime.IN:= TRUE;

			IF Popisovanie.IN.Laser_StavREADY AND Safety.STAV.ZonaLaser_Aktivna THEN
				SC_Popisovanie.ResetStep:= TRUE;
				SC_Popisovanie.Step:= 113;
			END_IF

			IF SC_Popisovanie.AlarmTime.Q THEN
				Alarmy[25]:= TRUE;
				PoruchaPopisovania:= TRUE;
				Zariadenie.KoniecCyklu:= TRUE;
			END_IF

		113:
			SC_Popisovanie.StepName:='113 - Automaticky Rezim - start popisovania';
			SC_Popisovanie.IdleTime.PT:= T#8s;
			SC_Popisovanie.AlarmTime.PT:= T#5s;

			IF NOT SC_Popisovanie.Switch1 THEN
				Popisovanie.OUT.Laser_StartZnacenia:= TRUE;
				SC_Popisovanie.Switch1:= TRUE;
			END_IF

			IF Popisovanie.IN.Laser_StavBUSY THEN
				Popisovanie.OUT.Laser_StartZnacenia:= FALSE;
				SC_Popisovanie.ResetStep:= TRUE;
				SC_Popisovanie.Step:= 114;
			END_IF

		114:
			SC_Popisovanie.StepName:='114 - Automaticky Rezim - cakam na ukoncenie popisovania';
			SC_Popisovanie.IdleTime.PT:= T#8s;
			SC_Popisovanie.AlarmTime.PT:= T#5s;

			IF Popisovanie.IN.Laser_StavEND THEN
				Stav_StatorPopisany:= TRUE;
				SC_Popisovanie.ResetStep:= TRUE;
				SC_Popisovanie.Step:= 115;
			END_IF

		115:
			SC_Popisovanie.StepName:='115 - Automaticky Rezim - zasunutie zdvizky';
			SC_Popisovanie.IdleTime.PT:= T#500ms;
			SC_Popisovanie.AlarmTime.PT:= T#5s;

			IF NOT SC_Popisovanie.Switch1 THEN
				Zdvizku_ZASUN:= TRUE;
				SC_Popisovanie.Switch1:= TRUE;
			END_IF

			IF Popisovanie.IN.Zdvizka_ZASUNUTA AND NOT Safety.STAV.SnimacStatorPodLaserom_Aktivny THEN
				SC_Popisovanie.ResetStep:= TRUE;
				SC_Popisovanie.Step:= 130;
			ELSIF Popisovanie.IN.Zdvizka_ZASUNUTA AND Safety.STAV.SnimacStatorPodLaserom_Aktivny THEN
				Alarmy[24]:= TRUE;
				PoruchaPopisovania:= TRUE;
				Zariadenie.KoniecCyklu:= TRUE;
			END_IF

		120:
			SC_Popisovanie.StepName:='120 - Automaticky Rezim - kontrola poctu prazdnych paletiek';
			SC_Popisovanie.IdleTime.PT:= T#8s;
			SC_Popisovanie.AlarmTime.PT:= T#5s;

			IF Popisovanie.PAR.PocetPrazdnychPaletiek >= 2 THEN
				Zariadenie.KoniecModelu:= TRUE;
				Vizu.Zobraz_HlasenieVymenaModelu:= 0;
				SC_Popisovanie.ResetStep:= TRUE;
				SC_Popisovanie.Step:= 130;
			ELSE
				SC_Popisovanie.ResetStep:= TRUE;
				SC_Popisovanie.Step:= 130;
			END_IF

		130:
			SC_Popisovanie.StepName:='130 - Automaticky Rezim - cakam na uvolnenie snimaca zasoby pred kamerou';
			SC_Popisovanie.IdleTime.PT:= T#200ms;
			SC_Popisovanie.AlarmTime.PT:= T#5s;

			SC_Popisovanie.IdleTime.IN:= NOT Checker.IN.ZasobaPredStoprom1;

			IF SC_Popisovanie.IdleTime.Q THEN
				SC_Popisovanie.ResetStep:= TRUE;
				SC_Popisovanie.Step:= 131;
			ELSIF Popisovanie.KoniecCyklu THEN
				SC_Popisovanie.ResetStep:= TRUE;
				SC_Popisovanie.Step:= 0;
			END_IF

		131:
			SC_Popisovanie.StepName:='131 - Automaticky Rezim - zasunutie stopra zdvizky';
			SC_Popisovanie.IdleTime.PT:= T#500ms;
			SC_Popisovanie.AlarmTime.PT:= T#5s;

			IF NOT SC_Popisovanie.Switch1 THEN
				StoperZdvizky_ZASUN:= TRUE;
				SC_Popisovanie.Switch1:= TRUE;
			END_IF

			IF Popisovanie.IN.StoperZdvizky_ZASUNUTY THEN
				Stav_StatorPopisany:= FALSE;
				SC_Popisovanie.ResetStep:= TRUE;
				SC_Popisovanie.Step:= 133;
			END_IF

		133:
			SC_Popisovanie.StepName:='133 - Automaticky Rezim - cakam na odchod paletky zo stopra zdvizky';
			SC_Popisovanie.IdleTime.PT:= T#500ms;
			SC_Popisovanie.AlarmTime.PT:= T#5s;

			SC_Popisovanie.IdleTime.IN:= NOT Popisovanie.IN.StoperZdvizky_PritomnostPaletky;

			IF SC_Popisovanie.IdleTime.Q THEN
				SC_Popisovanie.ResetStep:= TRUE;
				SC_Popisovanie.Step:= 135;
			END_IF

		135:
			SC_Popisovanie.StepName:='135 - Automaticky Rezim - vysunutie stopra zdvizky';
			SC_Popisovanie.IdleTime.PT:= T#500ms;
			SC_Popisovanie.AlarmTime.PT:= T#5s;

			IF NOT SC_Popisovanie.Switch1 THEN
				StoperZdvizky_VYSUN:= TRUE;
				SC_Popisovanie.Switch1:= TRUE;
			END_IF

			IF Popisovanie.IN.StoperZdvizky_VYSUNUTY THEN
				SC_Popisovanie.ResetStep:= TRUE;
				SC_Popisovanie.Step:= 100;
			END_IF

			//*******************************************************Manuálny režim*******************************************************************************//
		700:
			SC_Popisovanie.StepName:='700 - Manualny Rezim';
			SC_Popisovanie.IdleTime.PT:= T#8s;
			SC_Popisovanie.AlarmTime.PT:= T#5s;

	END_CASE

END_PROGRAM

PROGRAM _EXIT
	(* Insert code here *)

END_PROGRAM
```

#### Variables.var - Local variables
```iecst
VAR
	SC_OvlStopra : SequenceControlTyp;
	StoperZdvizky_VYSUN : BOOL;
	StoperZdvizky_ZASUN : BOOL;
	SC_OvlZdvizky : SequenceControlTyp;
	Zdvizku_VYSUN : BOOL;
	Zdvizku_ZASUN : BOOL;
	KodStatora_PoleUSINT : ARRAY[0..19] OF USINT;
	length : UDINT;
	PosledneZnaky : STRING[4]; (*Posledné 4 znaky zo vstupu*)
	i : USINT;
	Rok_PoleUSINT : ARRAY[0..3] OF USINT;
	Rok_STRING : STRING[4];
	Rok_Cislica1 : STRING[1];
	Rok_Cislica2 : STRING[1];
END_VAR
```

#### OvlStopra.st
```iecst
ACTION OvlStopra:

	//Volanie funkcie SequenceControl//
	SequenceControl(SC:= SC_OvlStopra);

	CASE SC_OvlStopra.Step OF

		0:
			SC_OvlStopra.StepName:= '0 - Nulovanie';
			StoperZdvizky_VYSUN:= FALSE;
			StoperZdvizky_ZASUN:= FALSE;
			Popisovanie.OUT.StoperZdvizky_VYSUN:= FALSE;
			Popisovanie.OUT.StoperZdvizky_ZASUN:= FALSE;
			IF SC_Popisovanie.Step <> 0 THEN
				SC_OvlStopra.ResetStep:= TRUE;
				SC_OvlStopra.Step:= 1;
			END_IF

		1:
			SC_OvlStopra.StepName:= '1 - Rozhodnutie o cinnosti';
			IF StoperZdvizky_VYSUN THEN
				SC_OvlStopra.Step:= 10;
			ELSIF StoperZdvizky_ZASUN THEN
				SC_OvlStopra.Step:= 20;
			END_IF

		10:
			SC_OvlStopra.StepName:= '10 - Vysunutie stopra';
			SC_OvlStopra.IdleTime.PT:= T#3s;
			SC_OvlStopra.AlarmTime.PT:= T#3s;

			IF Popisovanie.Automat THEN
				SC_OvlStopra.AlarmTime.IN:= TRUE;
			ELSE
				SC_OvlStopra.IdleTime.IN:= TRUE;
			END_IF

			IF NOT SC_OvlStopra.Switch1 THEN
				Popisovanie.OUT.StoperZdvizky_VYSUN:= TRUE;
				SC_OvlStopra.Switch1:= TRUE;
			END_IF

			IF SC_OvlStopra.AlarmTime.Q THEN
				Alarmy[15]:= TRUE;
				PoruchaPopisovania:= TRUE;
				Zariadenie.KoniecCyklu:= TRUE;
			END_IF

			IF Popisovanie.IN.StoperZdvizky_VYSUNUTY OR SC_OvlStopra.IdleTime.Q THEN
				SC_OvlStopra.ResetStep:= TRUE;
				SC_OvlStopra.Step:= 0;
			END_IF

		20:
			SC_OvlStopra.StepName:= '20 - Zasunutie stopra';
			SC_OvlStopra.IdleTime.PT:= T#3s;
			SC_OvlStopra.AlarmTime.PT:= T#3s;

			IF Popisovanie.Automat THEN
				SC_OvlStopra.AlarmTime.IN:= TRUE;
			ELSE
				SC_OvlStopra.IdleTime.IN:= TRUE;
			END_IF

			IF NOT SC_OvlStopra.Switch1 THEN
				Popisovanie.OUT.StoperZdvizky_ZASUN:= TRUE;
				SC_OvlStopra.Switch1:= TRUE;
			END_IF

			IF SC_OvlStopra.AlarmTime.Q THEN
				Alarmy[16]:= TRUE;
				PoruchaPopisovania:= TRUE;
				Zariadenie.KoniecCyklu:= TRUE;
			END_IF

			IF Popisovanie.IN.StoperZdvizky_ZASUNUTY OR SC_OvlStopra.IdleTime.Q THEN
				SC_OvlStopra.ResetStep:= TRUE;
				SC_OvlStopra.Step:= 0;
			END_IF

	END_CASE

END_ACTION
```

#### OvlZdvizky.st
```iecst
ACTION OvlZdvizky:

	//Volanie funkcie SequenceControl//
	SequenceControl(SC:= SC_OvlZdvizky);

	CASE SC_OvlZdvizky.Step OF

		0:
			SC_OvlZdvizky.StepName:= '0 - Nulovanie';
			Zdvizku_VYSUN:= FALSE;
			Zdvizku_ZASUN:= FALSE;
			//Popisovanie.OUT.Zdvizku_VYSUN:= FALSE;
			(*Popisovanie.OUT.Zdvizku_ZASUN:= FALSE;*)
			IF SC_Popisovanie.Step <> 0 THEN
				SC_OvlZdvizky.ResetStep:= TRUE;
				SC_OvlZdvizky.Step:= 1;
			END_IF

		1:
			SC_OvlZdvizky.StepName:= '1 - Rozhodnutie o cinnosti';
			IF Zdvizku_VYSUN THEN
				SC_OvlZdvizky.Step:= 10;
			ELSIF Zdvizku_ZASUN THEN
				SC_OvlZdvizky.Step:= 20;
			END_IF

		10:
			SC_OvlZdvizky.StepName:= '10 - Vysunutie zdvizky';
			SC_OvlZdvizky.IdleTime.PT:= T#3s;
			SC_OvlZdvizky.AlarmTime.PT:= T#3s;

			IF Popisovanie.Automat THEN
				SC_OvlZdvizky.AlarmTime.IN:= TRUE;
			ELSE
				SC_OvlZdvizky.IdleTime.IN:= TRUE;
			END_IF

			IF NOT SC_OvlZdvizky.Switch1 THEN
				Popisovanie.OUT.Zdvizku_ZASUN:= FALSE;
				Popisovanie.OUT.Zdvizku_VYSUN:= TRUE;
				SC_OvlZdvizky.IdleTime.IN:= TRUE;
				SC_OvlZdvizky.Switch1:= TRUE;
			END_IF

//			IF SC_OvlZdvizky.AlarmTime.Q THEN
//				Alarmy[17]:= TRUE;
//				PoruchaPopisovania:= TRUE;
//				Zariadenie.KoniecCyklu:= TRUE;
//			END_IF

			IF (Popisovanie.IN.Zdvizka_VYSUNUTA OR Safety.STAV.SnimacStatorPodLaserom_Aktivny) OR SC_OvlZdvizky.IdleTime.Q THEN
				SC_OvlZdvizky.ResetStep:= TRUE;
				SC_OvlZdvizky.Step:= 0;
			END_IF

		20:
			SC_OvlZdvizky.StepName:= '20 - Zasunutie zdvizky';
			SC_OvlZdvizky.IdleTime.PT:= T#3s;
			SC_OvlZdvizky.AlarmTime.PT:= T#3s;

			IF Popisovanie.Automat THEN
				SC_OvlZdvizky.AlarmTime.IN:= TRUE;
			ELSE
				SC_OvlZdvizky.IdleTime.IN:= TRUE;
			END_IF

			IF NOT SC_OvlZdvizky.Switch1 THEN
				Popisovanie.OUT.Zdvizku_VYSUN:= FALSE;
				Popisovanie.OUT.Zdvizku_ZASUN:= TRUE;
				SC_OvlZdvizky.Switch1:= TRUE;
			END_IF

			IF SC_OvlZdvizky.AlarmTime.Q THEN
				Alarmy[18]:= TRUE;
				PoruchaPopisovania:= TRUE;
				Zariadenie.KoniecCyklu:= TRUE;
			END_IF

			IF Popisovanie.IN.Zdvizka_ZASUNUTA OR SC_OvlZdvizky.IdleTime.Q THEN
				SC_OvlZdvizky.ResetStep:= TRUE;
				SC_OvlZdvizky.Step:= 0;
			END_IF

	END_CASE

END_ACTION
```

#### SpravaPreLaser.st
```iecst
ACTION SpravaPreLaser:

  //*********************************Položky ktoré obsahuje QR kód*********************************************************//
  	//*******BOM materiálu***********//
	QR_Kod.BOM_Statora:= ZvolenyBOM_kod_Statora;  //8 znakov

	//*******Dátum výroby************//
	//Deň//
	IF System_Cas_Datum.day < 10 THEN
		brsstrcpy(ADR(Systemovy_Datum_STR.Den),ADR('0'));
		Den_String:= USINT_TO_STRING(System_Cas_Datum.day);
		brsstrcat(ADR(Systemovy_Datum_STR.Den),ADR(Den_String));
	ELSE
		Systemovy_Datum_STR.Den:= USINT_TO_STRING(System_Cas_Datum.day);
	END_IF
	//Mesiac//
	IF System_Cas_Datum.month < 10 THEN
		brsstrcpy(ADR(Systemovy_Datum_STR.Mesiac),ADR('0'));
		Mesiac_String:= USINT_TO_STRING(System_Cas_Datum.month);
		brsstrcat(ADR(Systemovy_Datum_STR.Mesiac),ADR(Mesiac_String));
	ELSE
		Systemovy_Datum_STR.Mesiac:= USINT_TO_STRING(System_Cas_Datum.month);
	END_IF
    //Rok//
    Rok_STRING:= UINT_TO_STRING(System_Cas_Datum.year);
    brsmemcpy(ADR(Rok_PoleUSINT),ADR(Rok_STRING),SIZEOF(Rok_STRING));

    brsmemcpy(ADR(Rok_Cislica1),ADR(Rok_PoleUSINT[2]),SIZEOF(Rok_PoleUSINT[2]));
    brsmemcpy(ADR(Rok_Cislica2),ADR(Rok_PoleUSINT[3]),SIZEOF(Rok_PoleUSINT[3]));

    Systemovy_Datum_STR.Rok:= '';
    brsstrcat(ADR(Systemovy_Datum_STR.Rok),ADR(Rok_Cislica1));
    brsstrcat(ADR(Systemovy_Datum_STR.Rok),ADR(Rok_Cislica2));

	TextPole_Datum:='';
	brsstrcat(ADR(TextPole_Datum),ADR(Systemovy_Datum_STR.Rok));
    (*brsstrcat(ADR(TextPole_Datum),ADR(SeparatorDatumu));*)
    brsstrcat(ADR(TextPole_Datum),ADR(Systemovy_Datum_STR.Mesiac));
    (*brsstrcat(ADR(TextPole_Datum),ADR(SeparatorDatumu));*)
    brsstrcat(ADR(TextPole_Datum),ADR(Systemovy_Datum_STR.Den));

    QR_Kod.DatumVyroby:= TextPole_Datum;  //8 znakov

	//*********Čas výroby*************//
	//Hodina//
	IF System_Cas_Datum.hour < 10 THEN
		brsstrcpy(ADR(Systemovy_Cas_STR.Hodina),ADR('0'));
		Hodina_String:= USINT_TO_STRING(System_Cas_Datum.hour);
		brsstrcat(ADR(Systemovy_Cas_STR.Hodina),ADR(Hodina_String));
	ELSE
		Systemovy_Cas_STR.Hodina:= USINT_TO_STRING(System_Cas_Datum.hour);
	END_IF

	//Minúta//
	IF System_Cas_Datum.minute < 10 THEN
		brsstrcpy(ADR(Systemovy_Cas_STR.Minuta),ADR('0'));
		Minuta_String:= USINT_TO_STRING(System_Cas_Datum.minute);
		brsstrcat(ADR(Systemovy_Cas_STR.Minuta),ADR(Minuta_String));
	ELSE
		Systemovy_Cas_STR.Minuta:= USINT_TO_STRING(System_Cas_Datum.minute);
	END_IF

    //Sekunda//
    IF System_Cas_Datum.second < 10 THEN
        brsstrcpy(ADR(Systemovy_Cas_STR.Sekunda),ADR('0'));
        Sekunda_String:= USINT_TO_STRING(System_Cas_Datum.second);
        brsstrcat(ADR(Systemovy_Cas_STR.Sekunda),ADR(Sekunda_String));
    ELSE
        Systemovy_Cas_STR.Sekunda:= USINT_TO_STRING(System_Cas_Datum.second);
    END_IF

	TextPole_Cas:='';
	brsstrcat(ADR(TextPole_Cas),ADR(Systemovy_Cas_STR.Hodina));
	(*brsstrcat(ADR(TextPole_Cas),ADR(SeparatorCasu));*)
	brsstrcat(ADR(TextPole_Cas),ADR(Systemovy_Cas_STR.Minuta));
	brsstrcat(ADR(TextPole_Cas),ADR(Systemovy_Cas_STR.Sekunda));

	QR_Kod.CasVyroby:= TextPole_Cas;  //6 znakov

	//*************Číslo výrobnej linky***************//
	QR_Kod.NazovVyrobnejLinky:= 'StatorEM';   //8 znakov

	//**************Vyčítavanie posledných štyroch znakov z BOM materiálu**************//

	length := brsstrlen(ADR(ZvolenyBOM_kod_Statora)); //Zistí počet znakov//
	IF length >= 4 THEN
		brsmemcpy(ADR(KodStatora_PoleUSINT),ADR(ZvolenyBOM_kod_Statora),SIZEOF(ZvolenyBOM_kod_Statora));
		i := KodStatora_PoleUSINT[length-4];
		brsstrcpy(ADR(PosledneZnaky),ADR(i));
		i := KodStatora_PoleUSINT[length-3];
		brsstrcat(ADR(PosledneZnaky),ADR(i));
		i := KodStatora_PoleUSINT[length-2];
		brsstrcat(ADR(PosledneZnaky),ADR(i));
		i := KodStatora_PoleUSINT[length-1];
		brsstrcat(ADR(PosledneZnaky),ADR(i));
	END_IF

	QR_Kod.BOM_PosledneZnaky:= PosledneZnaky;  //4 znaky

	//***************************************Vytvorenie správy pre laser*******************************************

	brsmemcpy(ADR(Laser_DataSpravy[8]),ADR(QR_Kod.BOM_Statora),7);  			//Pole č.0
	brsmemcpy(ADR(Laser_DataSpravy[17]),ADR(QR_Kod.DatumVyroby),6);				//Pole č.1
	brsmemcpy(ADR(Laser_DataSpravy[25]),ADR(QR_Kod.CasVyroby),6);				//Pole č.2
	brsmemcpy(ADR(Laser_DataSpravy[33]),ADR(QR_Kod.NazovVyrobnejLinky),8);  	//Pole č.3
	brsmemcpy(ADR(Laser_DataSpravy[43]),ADR(QR_Kod.BOM_PosledneZnaky),4);       //Pole č.4

END_ACTION
```

### Program Logical/Program/Checker (IEC)

#### Main.st - Init, cyclic, exit code
```iecst
PROGRAM _INIT
	Checker.TRIGER_Enable:= TRUE;

END_PROGRAM

PROGRAM _CYCLIC

	//Volanie podprogramov//
	OvlStoprov;

	//Volanie funkcie SequenceControl//
	SequenceControl(SC:= SC_Checker);

	//Reset sekcie //
	IF Checker.Reset OR PoruchaCheckera THEN
		SC_Checker.Step:= 0;
	END_IF

	CASE SC_Checker.Step OF

		0:
			SC_Checker.StepName:='0 - Nulovanie';
			SC_OvlStoprov.Step:= 0;
			Checker.Automat:= FALSE;
			Checker.KoniecCyklu:= FALSE;
			Checker.Manual:= FALSE;
			Checker.Reset:= FALSE;
			Checker.STAV.PoINIT:= FALSE;
			Checker.OUT.BANNER_CervenaLED:= FALSE;
			Checker.OUT.BANNER_ZelenaLED:= FALSE;
			Checker.TRIGER:= FALSE;
			Checker.Vysledok_POTVRDENIE:= FALSE;
			Zariadenie.KoniecModelu:= FALSE;

			IF Safety.STAV.ZonaCS_Aktivna AND NOT PoruchaCheckera AND Zariadenie.IN.TlakVzduchu_OK THEN
				SC_Checker.ResetStep:= TRUE;
				SC_Checker.Step:= 1;
			END_IF

		1:
			SC_Checker.StepName:='1 - Cakam na spustenie vyroby';
			IF Checker.Automat THEN
				SC_Checker.Step:= 2;
			ELSIF Checker.Manual THEN
				SC_Checker.Step:= 700;
			END_IF

			//********************************************************Inicializácia****************************************************************************//

		2:
			SC_Checker.StepName:='2 - Inicializacia - cakam na spustenie inicializacie';
			SC_Checker.IdleTime.PT:= T#500ms;
			SC_Checker.AlarmTime.PT:= T#5s;

			SC_Checker.IdleTime.IN:= TRUE;

			IF SC_Checker.IdleTime.Q THEN
				SC_Checker.ResetStep:= TRUE;
				SC_Checker.Step:= 3;
			END_IF

		3:
			SC_Checker.StepName:='3 - Inicializacia - rozhodnutie o inicializacii';
			SC_Checker.IdleTime.PT:= T#500ms;
			SC_Checker.AlarmTime.PT:= T#5s;

			IF Checker.STAV.Stopre_PoziciaNAVAZANIE THEN
				(*Checker.OUT.BANNER_ZelenaLED:= TRUE;*)
				SC_Checker.ResetStep:= TRUE;
				SC_Checker.Step:= 10;
			ELSIF Checker.STAV.Stopre_PoziciaVYVAZANIE THEN
				SC_Checker.ResetStep:= TRUE;
				SC_Checker.Step:= 5;
			ELSE
				SC_Checker.ResetStep:= TRUE;
				SC_Checker.Step:= 7;
			END_IF

		5:
			SC_Checker.StepName:='5 - Inicializacia - cakam na odchod paletky z 2 stopra';
			SC_Checker.IdleTime.PT:= T#500ms;
			SC_Checker.AlarmTime.PT:= T#5s;

			SC_Checker.IdleTime.IN:= NOT Checker.IN.Stoper2_PritomnostPaletky;

			IF SC_Checker.IdleTime.Q THEN
				SC_Checker.ResetStep:= TRUE;
				SC_Checker.Step:= 7;
			END_IF

		7:
			SC_Checker.StepName:='7 - Inicializacia - preklopenie stoprov do pozicie navazania';
			SC_Checker.IdleTime.PT:= T#500ms;
			SC_Checker.AlarmTime.PT:= T#5s;

			IF NOT SC_Checker.Switch1 THEN
				Stopre_pozNAVAZANIE:= TRUE;
				SC_Checker.Switch1:= TRUE;
			END_IF

			IF Checker.STAV.Stopre_PoziciaNAVAZANIE THEN
				(*Checker.OUT.BANNER_ZelenaLED:= TRUE;*)
				SC_Checker.ResetStep:= TRUE;
				SC_Checker.Step:= 10;
			END_IF

		10:
			SC_Checker.StepName:='10 - Inicializacia - vynulovanie bitu novy vysledok checkera READY';
			SC_Checker.IdleTime.PT:= T#500ms;
			SC_Checker.AlarmTime.PT:= T#5s;

			IF Checker.STAV.Vysledok_READY THEN
				Checker.Vysledok_POTVRDENIE:= TRUE;
			ELSE
				Checker.Vysledok_POTVRDENIE:= FALSE;
				Checker.STAV.PoINIT:= TRUE;
				SC_Checker.ResetStep:= TRUE;
				SC_Checker.Step:= 100;
			END_IF

			//********************************************************Automatický režim****************************************************************************//

		100:
			SC_Checker.StepName:='100 - Automaticky Rezim - cakam na pritomnost paletky na 2 stopri';
			SC_Checker.IdleTime.PT:= T#1s;
			SC_Checker.AlarmTime.PT:= T#5s;

			SC_Checker.IdleTime.IN:= Checker.IN.Stoper2_PritomnostPaletky;
			SC_Checker.AlarmTime.IN:= NOT Checker.IN.Stoper2_PritomnostPaletky;

			IF SC_Checker.IdleTime.Q THEN
				SC_Checker.ResetStep:= TRUE;
				SC_Checker.Step:= 105;
			ELSIF Checker.KoniecCyklu AND NOT Popisovanie.Automat THEN
				SC_Checker.ResetStep:= TRUE;
				SC_Checker.Step:= 0;
			ELSIF Zariadenie.KoniecModelu AND SC_Checker.AlarmTime.Q THEN
				SC_Checker.ResetStep:= TRUE;
				SC_Checker.Step:= 0;
			END_IF

		105:
			SC_Checker.StepName:='105 - Automaticky Rezim - rozhodnutie o kontrole QR kodu';
			SC_Checker.IdleTime.PT:= T#500ms;
			SC_Checker.AlarmTime.PT:= T#5s;

			IF Zariadenie.PriechodnyRezim THEN
				SC_Checker.ResetStep:= TRUE;
				SC_Checker.Step:= 120;
			ELSIF Checker.KAMERA_OFF THEN
				SC_Checker.ResetStep:= TRUE;
				SC_Checker.Step:= 120;
			ELSIF Checker.IN.Stoper2_PritomnostStatora THEN
				SC_Checker.ResetStep:= TRUE;
				SC_Checker.Step:= 109;
			ELSE
				SC_Checker.ResetStep:= TRUE;
				SC_Checker.Step:= 120;
			END_IF

		109:
			SC_Checker.StepName:='10 - Automaticky Rezim - vynulovanie bitu novy vysledok checkera READY';
			SC_Checker.IdleTime.PT:= T#500ms;
			SC_Checker.AlarmTime.PT:= T#5s;

			IF Checker.STAV.Vysledok_READY THEN
				Checker.Vysledok_POTVRDENIE:= TRUE;
			ELSE
				Checker.Vysledok_POTVRDENIE:= FALSE;
				SC_Checker.ResetStep:= TRUE;
				SC_Checker.Step:= 110;
			END_IF

		110:
			SC_Checker.StepName:='110 - Automaticky Rezim - start citania QR kodu';
			SC_Checker.IdleTime.PT:= T#500ms;
			SC_Checker.AlarmTime.PT:= T#5s;

			IF NOT SC_Checker.Switch1 THEN
				Checker.TRIGER:= TRUE;
				SC_Checker.IdleTime.IN:= TRUE;
				SC_Checker.Switch1:= TRUE;
			END_IF

			IF Checker.STAV.BUSY OR SC_Checker.IdleTime.Q THEN
				Checker.TRIGER:= FALSE;
				SC_Checker.ResetStep:= TRUE;
				SC_Checker.Step:= 112;
			END_IF

		112:
			SC_Checker.StepName:='112 - Automaticky Rezim - cakam na vysledok z kamery';
			SC_Checker.IdleTime.PT:= T#500ms;
			SC_Checker.AlarmTime.PT:= T#5s;

			IF Checker.STAV.Vysledok_READY THEN
				IF Checker.STAV.Vysledok_OK THEN
					Checker.OUT.BANNER_CervenaLED:= FALSE;
					(*Checker.OUT.BANNER_ZelenaLED:= TRUE;*)
					SC_Checker.ResetStep:= TRUE;
					SC_Checker.Step:= 120;
				ELSIF Checker.STAV.Vysledok_NG THEN
					(*Checker.OUT.BANNER_ZelenaLED:= FALSE;*)
					SC_Checker.ResetStep:= TRUE;
					SC_Checker.Step:= 115;
				END_IF
			ELSIF Checker.KAMERA_OFF THEN
				SC_Checker.ResetStep:= TRUE;
				SC_Checker.Step:= 120;
			END_IF

		115:
			SC_Checker.StepName:='115 - Automaticky Rezim - vysunutie stopra 1';
			SC_Checker.IdleTime.PT:= T#1s;
			SC_Checker.AlarmTime.PT:= T#5s;

			IF NOT SC_Checker.Switch1 THEN
				Stoper1_VYSUN:= TRUE;
				SC_Checker.Switch1:= TRUE;
			END_IF

			IF Checker.IN.Stoper1_VYSUNUTY THEN
				SC_Checker.ResetStep:= TRUE;
				SC_Checker.Step:= 116;
			END_IF

		116:
			SC_Checker.StepName:='116 - Automaticky Rezim - cakam na odobratie statora s paletkou a potvrdenie bannerom';
			SC_Checker.IdleTime.PT:= T#1s;
			SC_Checker.AlarmTime.PT:= T#5s;

			Checker.OUT.BANNER_CervenaLED:= Blikac200ms;

			IF NOT Checker.IN.Stoper2_PritomnostPaletky AND NOT Checker.IN.Stoper2_PritomnostStatora AND Checker.IN.TlacitkoBANNER THEN
				Checker.OUT.BANNER_CervenaLED:= FALSE;
				(*Checker.OUT.BANNER_ZelenaLED:= TRUE;*)
				SC_Checker.ResetStep:= TRUE;
				SC_Checker.Step:= 117;
			ELSIF Checker.KoniecCyklu AND NOT Popisovanie.Automat THEN
				SC_Checker.ResetStep:= TRUE;
				SC_Checker.Step:= 0;
			END_IF

		117:
			SC_Checker.StepName:='117 - Automaticky Rezim - zasunutie stopra 1';
			SC_Checker.IdleTime.PT:= T#1s;
			SC_Checker.AlarmTime.PT:= T#5s;

			IF NOT SC_Checker.Switch1 THEN
				Stoper1_ZASUN:= TRUE;
				SC_Checker.Switch1:= TRUE;
			END_IF

			IF Checker.IN.Stoper1_ZASUNUTY THEN
				SC_Checker.ResetStep:= TRUE;
				SC_Checker.Step:= 100;
			END_IF

		120:
			SC_Checker.StepName:='120 - Automaticky Rezim - cakam na uvolnenie vystupnej trate';
			SC_Checker.IdleTime.PT:= T#1s;
			SC_Checker.AlarmTime.PT:= T#5s;

			SC_Checker.IdleTime.IN:= NOT Checker.IN.ZaplnenieVystupnejTrate;

			IF SC_Checker.IdleTime.Q THEN
				SC_Checker.ResetStep:= TRUE;
				SC_Checker.Step:= 121;
			ELSIF Checker.KoniecCyklu AND NOT Popisovanie.Automat THEN
				SC_Checker.ResetStep:= TRUE;
				SC_Checker.Step:= 0;
			END_IF

		121:
			SC_Checker.StepName:='121 - Automaticky Rezim - preklopenie stoprov do pozicie vyvazania';
			SC_Checker.IdleTime.PT:= T#500ms;
			SC_Checker.AlarmTime.PT:= T#5s;

			IF NOT SC_Checker.Switch1 THEN
				Stopre_pozVYVAZANIE:= TRUE;
				SC_Checker.Switch1:= TRUE;
			END_IF

			IF Checker.STAV.Stopre_PoziciaVYVAZANIE THEN
				Checker.STAV.PoINIT:= TRUE;
				SC_Checker.ResetStep:= TRUE;
				SC_Checker.Step:= 122;
			END_IF

		122:
			SC_Checker.StepName:='122 - Automaticky Rezim - cakam na odchod paletky z 2 stopra';
			SC_Checker.IdleTime.PT:= T#1s;
			SC_Checker.AlarmTime.PT:= T#5s;

			SC_Checker.IdleTime.IN:= NOT Checker.IN.Stoper2_PritomnostPaletky;

			IF SC_Checker.IdleTime.Q THEN
				SC_Checker.ResetStep:= TRUE;
				SC_Checker.Step:= 123;
			END_IF

		123:
			SC_Checker.StepName:='123 - Automaticky Rezim - preklopenie stoprov do pozicie navazania';
			SC_Checker.IdleTime.PT:= T#500ms;
			SC_Checker.AlarmTime.PT:= T#5s;

			IF NOT SC_Checker.Switch1 THEN
				Stopre_pozNAVAZANIE:= TRUE;
				SC_Checker.Switch1:= TRUE;
			END_IF

			IF Checker.STAV.Stopre_PoziciaNAVAZANIE THEN
				SC_Checker.ResetStep:= TRUE;
				SC_Checker.Step:= 100;
			END_IF

			//*******************************************************Manuálny režim*******************************************************************************//
		700:
			SC_Checker.StepName:='700 - Manualny Rezim';
			SC_Checker.IdleTime.PT:= T#8s;
			SC_Checker.AlarmTime.PT:= T#5s;

	END_CASE

END_PROGRAM

PROGRAM _EXIT
	(* Insert code here *)

END_PROGRAM
```

#### Variables.var - Local variables
```iecst
VAR
	SC_OvlStoprov : SequenceControlTyp;
	Stopre_pozNAVAZANIE : BOOL;
	Stopre_pozVYVAZANIE : BOOL;
	Stoper1_VYSUN : BOOL;
	Stoper1_ZASUN : BOOL;
END_VAR
```

#### OvlStoprov.st
```iecst
ACTION OvlStoprov:

	//Pozície stoprov//
	Checker.STAV.Stopre_PoziciaNAVAZANIE:= Checker.IN.Stoper1_ZASUNUTY AND Checker.IN.Stoper2_VYSUNUTY;
	Checker.STAV.Stopre_PoziciaVYVAZANIE:= Checker.IN.Stoper1_VYSUNUTY AND Checker.IN.Stoper2_ZASUNUTY;

	//Volanie funkcie SequenceControl//
	SequenceControl(SC:= SC_OvlStoprov);

	CASE SC_OvlStoprov.Step OF

		0:
			SC_OvlStoprov.StepName:= '0 - Nulovanie';
			Stopre_pozNAVAZANIE:= FALSE;
			Stopre_pozVYVAZANIE:= FALSE;
			Stoper1_VYSUN:= FALSE;
			Stoper1_ZASUN:= FALSE;
			Checker.OUT.Stoper1_VYSUN:= FALSE;
			Checker.OUT.Stoper1_ZASUN:= FALSE;
			Checker.OUT.Stoper2_VYSUN:= FALSE;
			Checker.OUT.Stoper2_ZASUN:= FALSE;
			IF SC_Checker.Step <> 0 THEN
				SC_OvlStoprov.ResetStep:= TRUE;
				SC_OvlStoprov.Step:= 1;
			END_IF

		1:
			SC_OvlStoprov.StepName:= '1 - Rozhodnutie o cinnosti';
			IF Stopre_pozNAVAZANIE THEN
				SC_OvlStoprov.Step:= 10;
			ELSIF Stopre_pozVYVAZANIE THEN
				SC_OvlStoprov.Step:= 20;
			ELSIF Stoper1_VYSUN THEN
				SC_OvlStoprov.Step:= 30;
			ELSIF Stoper1_ZASUN THEN
				SC_OvlStoprov.Step:= 40;
			END_IF

		10:
			SC_OvlStoprov.StepName:= '10 - Prepnutie oddelovaca do pozicie navazania';
			SC_OvlStoprov.IdleTime.PT:= T#3s;
			SC_OvlStoprov.AlarmTime.PT:= T#3s;

			IF Checker.Automat THEN
				SC_OvlStoprov.AlarmTime.IN:= TRUE;
			ELSE
				SC_OvlStoprov.IdleTime.IN:= TRUE;
			END_IF

			IF NOT SC_OvlStoprov.Switch1 THEN
				Checker.OUT.Stoper1_ZASUN:= TRUE;
				Checker.OUT.Stoper2_VYSUN:= TRUE;
				SC_OvlStoprov.Switch1:= TRUE;
			END_IF

			IF SC_OvlStoprov.AlarmTime.Q THEN
				IF NOT Checker.IN.Stoper1_ZASUNUTY THEN
					Alarmy[19]:= TRUE;
				ELSIF NOT Checker.IN.Stoper2_VYSUNUTY THEN
					Alarmy[22]:= TRUE;
				END_IF
				PoruchaCheckera:= TRUE;
				Zariadenie.KoniecCyklu:= TRUE;
			END_IF

			IF Checker.STAV.Stopre_PoziciaNAVAZANIE OR SC_OvlStoprov.IdleTime.Q THEN
				SC_OvlStoprov.ResetStep:= TRUE;
				SC_OvlStoprov.Step:= 0;
			END_IF

		20:
			SC_OvlStoprov.StepName:= '20 - Prepnutie oddelovaca do pozicie vyvazania';
			SC_OvlStoprov.IdleTime.PT:= T#3s;
			SC_OvlStoprov.AlarmTime.PT:= T#3s;

			IF Checker.Automat THEN
				SC_OvlStoprov.AlarmTime.IN:= TRUE;
			ELSE
				SC_OvlStoprov.IdleTime.IN:= TRUE;
			END_IF

			IF NOT SC_OvlStoprov.Switch1 THEN
				Checker.OUT.Stoper1_VYSUN:= TRUE;
				Checker.OUT.Stoper2_ZASUN:= TRUE;
				SC_OvlStoprov.Switch1:= TRUE;
			END_IF

			IF SC_OvlStoprov.AlarmTime.Q THEN
				IF NOT Checker.IN.Stoper1_VYSUNUTY THEN
					Alarmy[21]:= TRUE;
				ELSIF NOT Checker.IN.Stoper2_ZASUNUTY THEN
					Alarmy[20]:= TRUE;
				END_IF
				PoruchaCheckera:= TRUE;
				Zariadenie.KoniecCyklu:= TRUE;
			END_IF

			IF Checker.STAV.Stopre_PoziciaVYVAZANIE OR SC_OvlStoprov.IdleTime.Q THEN
				SC_OvlStoprov.ResetStep:= TRUE;
				SC_OvlStoprov.Step:= 0;
			END_IF

		30:
			SC_OvlStoprov.StepName:= '30 - Vysunutie stopra 1';
			SC_OvlStoprov.IdleTime.PT:= T#3s;
			SC_OvlStoprov.AlarmTime.PT:= T#3s;

			IF Checker.Automat THEN
				SC_OvlStoprov.AlarmTime.IN:= TRUE;
			ELSE
				SC_OvlStoprov.IdleTime.IN:= TRUE;
			END_IF

			IF NOT SC_OvlStoprov.Switch1 THEN
				Checker.OUT.Stoper1_VYSUN:= TRUE;
				SC_OvlStoprov.Switch1:= TRUE;
			END_IF

			IF SC_OvlStoprov.AlarmTime.Q THEN
				Alarmy[21]:= TRUE;
				PoruchaCheckera:= TRUE;
				Zariadenie.KoniecCyklu:= TRUE;
			END_IF

			IF Checker.IN.Stoper1_VYSUNUTY OR SC_OvlStoprov.IdleTime.Q THEN
				SC_OvlStoprov.ResetStep:= TRUE;
				SC_OvlStoprov.Step:= 0;
			END_IF

		40:
			SC_OvlStoprov.StepName:= '40 - Zasunutie stopra 1';
			SC_OvlStoprov.IdleTime.PT:= T#3s;
			SC_OvlStoprov.AlarmTime.PT:= T#3s;

			IF Checker.Automat THEN
				SC_OvlStoprov.AlarmTime.IN:= TRUE;
			ELSE
				SC_OvlStoprov.IdleTime.IN:= TRUE;
			END_IF

			IF NOT SC_OvlStoprov.Switch1 THEN
				Checker.OUT.Stoper1_ZASUN:= TRUE;
				SC_OvlStoprov.Switch1:= TRUE;
			END_IF

			IF SC_OvlStoprov.AlarmTime.Q THEN
				Alarmy[19]:= TRUE;
				PoruchaCheckera:= TRUE;
				Zariadenie.KoniecCyklu:= TRUE;
			END_IF

			IF Checker.IN.Stoper1_ZASUNUTY OR SC_OvlStoprov.IdleTime.Q THEN
				SC_OvlStoprov.ResetStep:= TRUE;
				SC_OvlStoprov.Step:= 0;
			END_IF

	END_CASE

END_ACTION
```

### Program Logical/Program/Poruchy_Signalizacie (IEC)
